# B&R Automation Studio project vibratorControlWithCurrentController (part 10)

#### local.typ - Local data types
```iecst
TYPE
	local_no_opcua_typ : 	STRUCT
		configOld : config_vibrator_typ;
		recipeOld : recipe_vibrator_typ;
		configTmp : config_vibrator_typ;
		axisAlarmText : STRING[363];
		alarm : local_alarm_typ;
		TON_alarmReaction : TON;
		calibration : local_no_opcua_calibration_typ;
	END_STRUCT;
	local_no_opcua_calibration_typ : 	STRUCT
		maxAmplitude : REAL;
		maxVibration : REAL;
		stepSizeAmplitude : REAL;
		tmpAmplitude : REAL;
		counter : USINT;
		bufferIdx : UINT;
		countTestPulse : USINT;
		boostCaliDone : BOOL;
		breakCaliDone : BOOL;
		countPulsesToFinetune : USINT;
	END_STRUCT;
	local_typ : 	STRUCT
		recipeName : STRING[80];
		configName : STRING[80];
		recipeNameCurrent : STRING[80];
		calibration : calibration_typ;
		MpRecipeRegPar_Config : MpRecipeRegPar;
		MpRecipeRegPar_Recipe : MpRecipeRegPar;
		MpRecipeRegPar_RecipeCurrent : MpRecipeRegPar;
		time : local_time_typ;
		MTBasicsLimiter_0 : MTBasicsLimiter;
		MC_BR_WriteParID_0 : MC_BR_WriteParID;
		vibAmplitude : REAL;
		highSpeed : BOOL;
		vibPercentAmplitude : REAL; (*amplitude for P3*)
		oldVibPercentAmplitude : REAL;
		vibAcceleration : REAL;
		sweep : local_sweep_typ;
		hmi : hmi_typ;
		vibFrequency : REAL := 50; (*[Hz] Frequency of virator*)
		calibrateState : UDINT;
		rampUp : REAL;
		linearizationSweep : linearizationSweep_typ;
		hw : local_hw_typ;
		linearizationTable : MTLookUpTable;
		lookUpFrequency : MTLookUpTable;
		pointsInLinearization : USINT;
		testAmplitude : BOOL;
		testDefault : BOOL;
		verifyLinearization : ARRAY[0..9]OF REAL;
		verifyIdx : USINT;
		testPercent : BOOL;
		oldSpeed : LEGO_SPEED_ENUM;
		oldCheckChangesConfig : BOOL;
		oldCheckChangesRecipe : BOOL;
		oldLoaded : BOOL;
		oldLoadedRecipe : BOOL;
		minimumTimeInCount : UDINT := 60000;
		DTGetTime_0 : DTGetTime;
		stateSimuPulse : USINT;
		simuTimeInCountSpeed : UDINT := 1000000;
		simuTimeInWaitSpeed : UDINT := 500000;
		simuTimeInStopped : UDINT := 600000;
		testProdFlow : BOOL;
		TON_delay : TON;
		currentAcceleration : REAL;
	END_STRUCT;
	calibration_typ : 	STRUCT
		TON_0 : TON;
		maxFreq : REAL;
		analogVib : REAL;
		sweepAmpl1CF : REAL := 0.5;
		sweepAmpl2CF : REAL := 0.6;
		sweepAmpl3CF : REAL := 1.0;
		sweepAmpl1LF : REAL := 0.09;
		sweepAmpl2LF : REAL := 0.08;
		sweepAmpl3LF : REAL := 0.11;
		sweepAmpl1LFbig : REAL := 0.1;
		sweepAmpl2LFbig : REAL := 0.08;
		sweepAmpl3LFbig : REAL := 0.11;
		sweepAmpl1CFbig : REAL := 1.7;
		sweepAmpl2CFbig : REAL := 1.4;
		sweepAmpl3CFbig : REAL := 1.8;
		timeToGetVibrWarm : TIME := T#11s;
		maxFreqFastSweep : REAL;
		bypassWarmUp : BOOL;
		slope : REAL;
		minAcceleration : REAL;
		minAccelerationTime : REAL;
		minAccelerationPhaseVelocity : REAL;
		accelerationStart : REAL;
		minAccelerationStart : REAL;
		freqBrakeCaliOffset : REAL;
		minFrequency : REAL;
		accelerationEnd : REAL;
		startBrakeFrequency : REAL;
	END_STRUCT;
	hmi_calibrate_typ : 	STRUCT
		activate : BOOL;
		calibrationToolPlugged : BOOL;
		progress : USINT;
		percentValue : REAL;
		testBoost : BOOL;
		enableStopButton : BOOL;
		runTestPulses : BOOL;
		increaseBoost : BOOL;
		increaseBrake : BOOL;
		decreaseBoost : BOOL;
		decreaseBrake : BOOL;
		enableBoostBrakeAdjustment : BOOL;
	END_STRUCT;
	linearizationSweep_typ : 	STRUCT
		actVibOld : REAL;
		sweepIdx : USINT;
		stableTime_TON : TON;
		a : REAL; (*Slope of linear function*)
		b : REAL; (*Intersection with y-axis in linear function*)
		MTBasicsPID_0 : MTBasicsPID;
		countStableSamples : USINT; (*If signal is less than allowed control error count one up.*)
		actIsOverSetValue : BOOL; (*True if act value is over set value.*)
		dcBusVoltage : REAL;
		supplyType : USINT; (*0=230V, 0=110V (Mexico)*)
	END_STRUCT;
	force_hw_typ : 	STRUCT
		enable : BOOL;
		current : REAL;
	END_STRUCT;
	hmi_typ : 	STRUCT
		config : config_vibrator_typ;
		calibratingProcessing : BOOL;
		cancelTuning : BOOL;
		recipe : recipe_vibrator_typ;
		calibration : hmi_calibrate_typ;
		force : force_hw_typ;
		needLinearization : BOOL;
		linearizationProcessing : BOOL;
		stopSweep : BOOL;
		oldCfType : SINT;
		actVoltage : REAL;
		targetAcceleration : REAL;
		voltage10Percent : REAL;
		voltage100Percent : REAL;
		recipeCurrent : recipe_vibrator_typ;
		waitSpeedLastBrick : USINT := 5;
		confirmPct : BOOL;
		increaseVibAmplitude : BOOL;
		decreaseVibAmplitude : BOOL;
		increaseVibAmplitudeFast : BOOL;
		decreaseVibAmplitudeFast : BOOL;
		linearizationGoalValue : REAL;
		enableOperatorInput : BOOL;
		showErrorMsgLinearization : BOOL;
		stopLinearization : BOOL;
		fitPercentTooLow : BOOL;
		linearizationActValue : REAL;
		daysSinceCalibration : REAL;
	END_STRUCT;
	local_time_typ : 	STRUCT
		elapsed : UDINT;
		maximum : UDINT;
	END_STRUCT;
	config_vibrator_typ : 	STRUCT
		tuneOnStartup : BOOL;
		vibFrequency : REAL := 50000;
		maxCurrent : REAL := 2.4;
		maxVoltage : REAL := 200;
		type : SINT; (*0=small CF, 1=big CF*)
		linearizationNodeVectorX : ARRAY[0..49]OF REAL;
		linearizationFcnValues : ARRAY[0..49]OF REAL;
		linearizationAccValues : ARRAY[0..49]OF REAL;
		linearizationFrequency1 : REAL; (*First frequency used for linear function for "voltage,frequency"*)
		linearizationFrequency2 : REAL; (*Second frequency used for linear function for "voltage,frequency"*)
		linearizationVoltage1 : REAL; (*First voltage used for linear function*)
		linearizationVoltage2 : REAL; (*Second voltage used for linear function*)
		pointY1 : REAL := 14;
		pointX1 : REAL := 10;
		pointY2 : REAL := 105;
		pointX2 : REAL := 100;
		Gain : REAL := 0.2;
		IntegrationTime : REAL := 1.5;
		minOut : REAL := 20;
		maxOut : REAL := 200;
		stableWindowPercent : REAL := 0.015;
		linearizeUsing3Points : BOOL := TRUE; (*True = only use 10%,55%,100% for linearization. *)
		frequencyVaryMode : BOOL := TRUE; (*This mode will vary the frequency depending on amplitude used on vibrator*)
		linearizationPercent : ARRAY[0..MAX_LOOKUP_POINTS]OF REAL;
		linearizationCurrent : ARRAY[0..MAX_LOOKUP_POINTS]OF REAL; (*Current at different percentages*)
		linearizationFrequencies : ARRAY[0..MAX_LOOKUP_POINTS]OF REAL; (*Frequency at different amplitudes*)
		linearizationAmplitude : ARRAY[0..MAX_LOOKUP_POINTS]OF REAL; (*Amplitude [A]*)
		fitPercentage : REAL; (*R^2 coefficient*)
		verifyLinearization : ARRAY[0..9]OF REAL;
		linearizationAccValue10pct : REAL;
		linearizationAccValue55pct : REAL;
		linearizationAccValue100pct : REAL;
		amplitudeFineTuning : REAL; (*This value will be add/subtract to the amplitude linearization result in case the calibration is a little off.*)
		emptyPercent : REAL;
		minimumTimeInCount : UDINT := 60000;
		calibrationDateTime : DATE_AND_TIME;
		boostVelocityLow : REAL;
		boostVelocityHigh : REAL;
		brakePhaseShiftVelocity : REAL;
		boostPhaseShiftVelocity : REAL;
		brakeVelocity : REAL;
		boostFrequency : REAL;
		brakeFrequency : REAL;
		boostAmplitude : REAL;
		brakeAmplitude : REAL;
		autoLinearizationAccAtCurrent : ARRAY[0..MAX_IDX_AUTO_LINEARIZATION]OF REAL;
		autoLinearizationCurrent : ARRAY[0..MAX_IDX_AUTO_LINEARIZATION]OF REAL;
		caliPulseBufferAcc : ARRAY[0..MAX_BUFFER_CALI_IDX]OF USINT;
		caliPulseEstimatedPct : ARRAY[0..MAX_BUFFER_CALI_IDX]OF USINT;
		disableLFBoost : BOOL;
	END_STRUCT;
	recipe_vibrator_typ : 	STRUCT
		waitSpeed : USINT := 10; (*%*)
		countingSpeed : USINT := 30; (*%*)
		rampUp : INT := 0; (*Time for 0 to 100 percent in msec*)
		useWaitSpeedCountingLastElement : BOOL := FALSE; (*If portion >2 and this is TRUE the vibrators will use waitSpeed when counting the last element, but belt will still keep counting speed.*)
	END_STRUCT;
	local_alarm_typ : 	STRUCT
		axisError : gAlarm_struct_typ;
	END_STRUCT;
	local_sweep_typ : 	STRUCT
		start : BOOL;
		amplitudeCFsmall : REAL := 0.8;
		amplitudeCFlarge : REAL := 1.2;
		amplitudeLF : REAL := 0.1;
		MTDataMinMax_0 : MTDataMinMax;
		frequencyStart : REAL := 48.5;
		frequencyStop : REAL := 50.4;
		maxVibrationISO : REAL;
		maxVibration : REAL;
		freqChangeRate : REAL := 0.02;
	END_STRUCT;
	local_hw_typ : 	STRUCT
		actVib : REAL;
		toggleBit : BOOL; (*Toggle bit will be true when we have new data ready*)
		ISO : REAL;
		analogInput : REAL;
		do_isBigCF : BOOL;
	END_STRUCT;
	axis_typ : 	STRUCT
		cmd : axis_cmd_typ;
		status : axis_status_typ;
		internal : axis_internal_typ;
	END_STRUCT;
	axis_cmd_typ : 	STRUCT
		power : BOOL;
	END_STRUCT;
	axis_status_typ : 	STRUCT
		powerOn : BOOL;
	END_STRUCT;
	axis_internal_typ : 	STRUCT
		MC_Power_0 : MC_Power;
	END_STRUCT;
	hmi_em_status_typ : 	STRUCT
		state : brdk_em_states_typ;
		substate : STRING[BRDK_MU_MAX_DESCRIPTION_STRING];
	END_STRUCT;
END_TYPE
```

#### local.var - Local variables
```iecst
VAR CONSTANT
	STATOR_RESISTANCE_SMALL_CF : REAL := 4.12;
	STATOR_RESISTANCE_SMALL_LF : REAL := 150;
	STATOR_INDUCTANCE_SMALL_CF : REAL := 0.230;
	STATOR_INDUCTANCE_SMALL_LF : REAL := 3.73;
	STATOR_RESISTANCE_BIG_CF : REAL := 4.96;
	STATOR_RESISTANCE_BIG_LF : REAL := 148.7;
	STATOR_INDUCTANCE_BIG_CF : REAL := 0.3;
	STATOR_INDUCTANCE_BIG_LF : REAL := 3.92;
	MAX_BUFFER_CALI_IDX : UINT := 399;
	VIBRATOR_FREQ_OFFSET : REAL := 0.1;
	VIBRATOR_FREQ_OFFSET_BIG_CF : REAL := 0.05;
END_VAR
VAR
	recipe : REFERENCE TO recipe_vibrator_typ;
	config : REFERENCE TO config_vibrator_typ;
	configTmp : REFERENCE TO config_vibrator_typ;
	em : REFERENCE TO brdkEM;
	i : UINT;
	j : USINT;
	k : UINT;
	localVariables : ARRAY[0..NUM_VIBRATOR] OF local_typ;
	localModule : ARRAY[0..NUM_VIBRATOR] OF brdkEM;
	this : REFERENCE TO local_typ;
	interface : REFERENCE TO gVibratorInterface_typ;
	watchIdx : USINT;
	axis : REFERENCE TO brdkMcBasic;
	localAxis : ARRAY[0..NUM_VIBRATOR] OF brdkMcBasic;
END_VAR
VAR CONSTANT
	MAX_IDX_AUTO_LINEARIZATION : USINT := 19;
	MAX_LOOKUP_POINTS : USINT := 4;
	SINE_WAVE_GENERATOR : UINT := 8752;
	CONTROLLER_MODE : UINT := 5;
	RATIO_ISO_TO_MAXPEAK : REAL := 95; (*Ration from ISO -> maxPeak (accelerometer value)*)
END_VAR
VAR
	em_status : ARRAY[0..NUM_VIBRATOR] OF hmi_em_status_typ;
	local : REFERENCE TO local_no_opcua_typ;
	local_no_opcua : ARRAY[0..NUM_VIBRATOR] OF local_no_opcua_typ;
END_VAR
```

#### LocalFunctions.fun
```iecst
{REDUND_ERROR} FUNCTION RSquared : REAL (*TODO: Add your comment here*) (*$GROUP=User,$CAT=User,$GROUPICON=User.png,$CATICON=User.png*)
	VAR_INPUT
		data : ARRAY[0..9] OF REAL;
		prc10 : REAL;
		prc100 : REAL;
	END_VAR
	VAR
		i : USINT;
		ssTot : REAL;
		ssRes : REAL;
		mean : REAL;
	END_VAR
END_FUNCTION

FUNCTION maxPeakToPercent : REAL
	VAR_INPUT
		maxPeakVal : REAL;
		Y1 : REAL;
		Y2 : REAL;
	END_VAR
	VAR
		slope : REAL;
	END_VAR
END_FUNCTION

FUNCTION getAccelerationFromPercent : REAL
	VAR_INPUT
		percent : REAL;
		vibratorType : UINT; (*0=CF, 1=LF*)
		machineType : SINT; (*0=small, 1=big*)
	END_VAR
END_FUNCTION
```

#### LocalFunctions.st
```iecst
FUNCTION RSquared
	mean := 0;
	FOR i:=0 TO 9 DO
		mean := mean + data[i];
	END_FOR
	mean := mean / 10;
	ssTot := 0;
	FOR i:=0 TO 9 DO
		ssTot := ssTot + pow(data[i]-mean, 2);
	END_FOR
	ssRes := 0;
	FOR i:=0 TO 9 DO
		ssRes := ssRes + pow(data[i]-(prc10+(((prc100-prc10)/9)*USINT_TO_REAL(i))), 2);
	END_FOR
	RSquared := 1 - (ssRes/ssTot);
END_FUNCTION

FUNCTION maxPeakToPercent
	IF (Y2-Y1) <> 0 THEN
		slope := 90/(Y2-Y1);
		maxPeakToPercent := LIMIT(0,slope*maxPeakVal+(10-(slope*Y1)),200);
	END_IF
END_FUNCTION

FUNCTION getAccelerationFromPercent

	IF machineType=0 THEN
		IF vibratorType=0 THEN
			// 10%=2756 , 100%=17420
			getAccelerationFromPercent := percent*162.93+1126.7;
		ELSE
			// 10%=1300 , 100%=10140
			getAccelerationFromPercent := percent*98.222+317.78;
		END_IF
	ELSE
		IF vibratorType=0 THEN
			// 10%=1456 , 100%=8060
			getAccelerationFromPercent := percent*73.378+722.22;
		ELSE
			// 10%=1508 , 100%=8840
			getAccelerationFromPercent := percent*81.467+693.33;
		END_IF
	END_IF

END_FUNCTION
```

### vibratorGlobal.typ
```iecst
TYPE
	gVibratorInterface_typ : 	STRUCT
		cmd : gVibratorInterface_cmd_typ;
		parameter : gVibratorInterface_parameter_typ;
		status : gVibratorInterface_status_typ;
	END_STRUCT;
	gVibratorInterface_cmd_typ : 	STRUCT
		speed : LEGO_SPEED_ENUM;
		calibrate : BOOL;
		copyRecipe : copy_recipe_command_typ;
		useWaitSpeed : BOOL; (*belt -> vibrator . Use waitSpeed even though belt is using countSpeed.*)
		monitorHighestAmplitude : BOOL; (*Will monitor highest analog acc value on accelerometer.*)
		readCurrentAndVoltage : BOOL;
		monitorActPeakValue : BOOL;
		monitorMaxPeakValue : BOOL;
		calibrationDone : BOOL;
		testPulses : BOOL;
		emptyPercent : REAL;
		reduceCountspeedWith5 : BOOL;
		runManualTest : BOOL;
		putRecipeForStalkElement : BOOL;
		initRecipe : BOOL;
		setCfType : BOOL;
	END_STRUCT;
	gVibratorInterface_parameter_typ : 	STRUCT
		speedPctManualTest : REAL;
		machineSize : USINT; (*0=Small CM, 1=Big CM*)
		CFType : USINT;
	END_STRUCT;
	gVibratorInterface_status_typ : 	STRUCT
		start : BOOL;
		calibrationDone : BOOL;
		calibratingMode : BOOL;
		machineType : SINT; (*0=small CM20, 1=big CM20*)
		highestAmplitudeAnalog : REAL;
		highestAmplitudeISO : REAL;
		highestAmplitudePeak : REAL;
		highestFrequencyAnalog : REAL;
		highestFrequencyISO : REAL;
		highestFrequencyPeak : REAL;
		highestAmplitude : REAL;
		highestFrequency : REAL;
		New_Member : USINT;
		actCurr : REAL;
		maxPeakValue : REAL;
		waitSpeed : USINT;
		countingSpeed : USINT;
		vibFrequency : REAL;
		vibAmplitude : REAL;
		vibAmplitudePercent : REAL;
		forcing : BOOL;
		percent : REAL;
		linearizationAmplitude : ARRAY[0..4]OF REAL;
		linearizationFrequencies : ARRAY[0..4]OF REAL;
		powered : BOOL;
		currAccelerometerPercent : REAL;
		currAccelerometerValue : REAL;
		calibrateBoost : BOOL;
		calibrateBrake : BOOL;
		brakePhaseShiftVelocity : REAL;
		boostPhaseShiftVelocity : REAL;
		minAccelerationStart : REAL;
		minAcceleration : REAL;
		minAccelerationTime : REAL;
		boostFrequency : REAL;
		brakeFrequency : REAL;
		brakeVelocity : REAL;
		boostVelocityLow : REAL;
		boostVelocityHigh : REAL;
		caliBoostVelocityLow : REAL;
		caliBoostVelocityHigh : REAL;
		calibrateBraketime : REAL;
		calibrateBrakeAmplitudeEnd : REAL;
		calibrateBrakeFrequencyEnd : REAL;
		boostAmpltiude : REAL;
		brakeAmplitude : REAL;
		caliProdTest : BOOL;
		currEstimatedPercent : REAL;
		isBigCF : BOOL;
		maxBoostPercent : REAL;
		minBreakPercent : REAL;
		filteredAccelerometerPercent : REAL;
		disableLFBoost : BOOL;
		rampUp : INT;
		calibrationResultFrequency : REAL;
		calibrationResultCurrent : REAL;
		calibrationResultCurrentOK : BOOL;
		calibrationResultFrequencyOK : BOOL;
		calibrationResultsReady : BOOL;
	END_STRUCT;
END_TYPE
```

### vibratorGlobal.var
```iecst
VAR
	gVibratorInterface : ARRAY[0..NUM_VIBRATOR] OF gVibratorInterface_typ;
END_VAR
VAR CONSTANT
	VIBRATOR_ALARM_SIZE : USINT := 0;
	NUM_VIBRATOR : USINT := 1; (*1 means 2*)
END_VAR
```

### Program Logical/modules/main/belt/belt (IEC)

#### producing.st
```iecst
ACTION producing:

	CASE em.state OF

		STATE_ACTIVATING:

			CASE em.substate OF

				0:
					IF (gRecipe.status.saved OR gRecipe.status.loaded) AND (gConfig.status.saved OR gConfig.status.loaded) THEN
						em.substate := 10;
					END_IF

				10:
					// Wait 20ms to make sure recipe is in the global variable. (belt in faster cyclic than vibrator)

					this.timeMinInCount := this.timeMinInCount + em.status.cycleTime;
					IF this.timeMinInCount > 20000 THEN
						this.timeMinInCount := 0;
						// Load CF/LF countspeed from recipe
						CFCountSpeed := gVibratorInterface[0].status.countingSpeed;
						LFCountSpeed := gVibratorInterface[1].status.countingSpeed;
						interface.status.recipeLoaded := TRUE;
						em.substate := 20;
					END_IF

				20:
					em.cmd.sc := TRUE;

			END_CASE

		STATE_STOPPED:
			em.description 	:= 'Waiting for start command';

			IF gConfig.status.loadInitialValue[2] AND (gRecipe.status.saved OR gRecipe.status.loaded) AND (gConfig.status.saved OR gConfig.status.loaded) THEN
				gConfig.status.loadInitialValue[2] := FALSE;
				recipe.countingSpeed := 300;
				recipe.useWaitSpeed := TRUE;
				recipe.waitSpeed := 110;
				recipe.rampUp := 50;
				recipe.rampDown := 30;
				recipe.itemGap := FALSE;
			END_IF

			// This case ONLY used for FAT
			CASE em.substate OF

				0:
					em.description := 'Wait for command';

					IF interface.cmd.doPhotoSensorTest THEN
						interface.status.photoSensorTestResult := TEST_NOT_DONE;
						this.hmi.statusFAT.torqueTestMaxProgress := 12000;
						this.hmi.statusFAT.torqueTestProgress := 0;
						this.hmi.statusFAT.photoSensorTestProgress := 0;
						this.hmi.statusFAT.photoSensorTestActive := TRUE;

						em.substate := 10;
					ELSIF interface.cmd.doPhotoSensorTestNoBelt THEN
						interface.cmd.doPhotoSensorTestNoBelt := FALSE;
						interface.status.photoSensorTestNoBeltResult := TEST_NOT_DONE;
						this.hmi.statusFAT.photoSensorTestNoBeltRunning := TRUE;
						this.timeElapsed := 0;
						em.substate := 50;
					END_IF

				10:
					em.description := 'Start servo and wait until it is running';

					interface.cmd.runManualTest := TRUE;
					interface.parameter.speedManualTest := 400;

//					IF this.hmi.cmd.stopPhotoSensorTest THEN	// stop cmd from user.
//						this.hmi.cmd.stopPhotoSensorTest := FALSE;
//						interface.status.photoSensorTestResult := TEST_STOPPED;
//						interface.cmd.startBelt := FALSE;
//						interface.par.beltSpeed := 0;
//						interface.cmd.doPhotoSensorTest := FALSE;
//						this.photoSensorTestProgress := 0;
//						this.hmi.status.photoSensorTestActive := FALSE;
//						em.substate := 0;
					IF axis.status.inMotion AND ABS(axis.status.actVelocity) > (interface.parameter.speedManualTest-50) THEN	// axis is running
						this.hmi.statusFAT.photoSensorTestProgress := 0;
						this.TON_photoSensorTest.PT := T#12000ms;
						this.TON_photoSensorTest.IN := FALSE;
						this.TON_photoSensorTest();
						// read parid for motor torque
						this.MC_BR_ReadParID_277.Axis := ADR(gAxisBelt);
						this.MC_BR_ReadParID_277.ParID := 277;
						this.MC_BR_ReadParID_277.DataType := ncPAR_TYP_REAL;
						this.MC_BR_ReadParID_277.DataAddress := ADR(this.motorTorque);
						this.MTDataMean_torque.Enable := TRUE;
						this.MTDataMean_torque.Reset := FALSE;
						this.MTDataMean_torque();

						em.substate := 11;
					END_IF

				11:
					em.description := 'Running photoSensor test';
					this.TON_photoSensorTest.IN := TRUE;
					// progress
					this.hmi.statusFAT.photoSensorTestProgress := TIME_TO_REAL(this.TON_photoSensorTest.ET);

					// read motor torque while running test.
					this.MC_BR_ReadParID_277.Execute := TRUE;
					this.MC_BR_ReadParID_277.Axis := ADR(gAxisBelt);
					this.MC_BR_ReadParID_277.DataAddress := ADR(this.motorTorque);

					IF this.MC_BR_ReadParID_277.Done THEN
						this.MC_BR_ReadParID_277.Execute := FALSE;
					END_IF
					this.MC_BR_ReadParID_277();
					IF this.hmi.statusFAT.photoSensorTestProgress >= 2500 THEN
						this.MTDataMean_torque.Reset := TRUE;
						this.MTDataMean_torque.In := ABS(this.motorTorque);
					END_IF
					this.MTDataMean_torque();

//					IF this.hmi.cmd.stopPhotoSensorTest THEN	// stop cmd from user.
//						this.hmi.cmd.stopPhotoSensorTest := FALSE;
//						this.TON_photoSensorTest.IN := FALSE;
//						interface.status.photoSensorTestResult := TEST_STOPPED;
//						interface.cmd.startBelt := FALSE;
//						interface.par.beltSpeed := 0;
//						interface.cmd.doPhotoSensorTest := FALSE;
//						this.photoSensorTestProgress := 0;
//						this.hmi.status.photoSensorTestActive := FALSE;
//						this.MTDataMean_torque(Enable:=FALSE,Reset:=FALSE);
//						em.substate := 15;
					IF this.hw.di_photo THEN
						interface.status.photoSensorTestResult := TEST_NOT_OK;
						this.TON_photoSensorTest.IN := FALSE;
						interface.cmd.runManualTest := FALSE;
						interface.parameter.speedManualTest := 0;
						this.hmi.avgMotorTorque := this.MTDataMean_torque.Out;
						interface.cmd.doPhotoSensorTest := FALSE;
						this.hmi.statusFAT.photoSensorTestProgress := 0;
						this.hmi.statusFAT.photoSensorTestActive := FALSE;
						this.MTDataMean_torque(Enable:=FALSE,Reset:=FALSE);
						em.substate := 15;
					ELSIF this.TON_photoSensorTest.Q THEN		// TODO: distanceConveyorShouldRun=6000 is random. How long should it run??
						IF this.MTDataMean_torque.Out < 0.25 THEN
							interface.status.photoSensorTestResult := TEST_OK;
							this.TON_photoSensorTest.IN := FALSE;
							interface.cmd.runManualTest := FALSE;
							interface.parameter.speedManualTest := 0;
							this.hmi.avgMotorTorque := this.MTDataMean_torque.Out;
							this.MTDataMean_torque(Enable:=FALSE,Reset:=FALSE);
							interface.cmd.doPhotoSensorTest := FALSE;
							this.hmi.statusFAT.photoSensorTestActive := FALSE;
							em.substate := 15;
						ELSE
							interface.status.photoSensorTestResult := TEST_NOT_OK;
							this.TON_photoSensorTest.IN := FALSE;
							interface.cmd.runManualTest := FALSE;
							this.hmi.avgMotorTorque := this.MTDataMean_torque.Out;
							interface.parameter.speedManualTest := 0;
							interface.cmd.doPhotoSensorTest := FALSE;
							this.hmi.statusFAT.photoSensorTestProgress := 0;
							this.hmi.statusFAT.photoSensorTestActive := FALSE;
							this.MTDataMean_torque(Enable:=FALSE,Reset:=FALSE);
							em.substate := 15;
						END_IF
					END_IF
					this.TON_photoSensorTest();

				15:
					em.description := 'Wait for readParId to be done (not busy)';

					this.MC_BR_ReadParID_277.Execute := FALSE;
					this.MC_BR_ReadParID_277.Axis := ADR(gAxisBelt);
					this.MC_BR_ReadParID_277.DataAddress := ADR(this.motorTorque);
					this.MC_BR_ReadParID_277();

					IF NOT this.MC_BR_ReadParID_277.Busy THEN
						em.substate := 0;
					END_IF

				50:
					em.description := 'Photo sensor test with no belt';

					this.timeElapsed := this.timeElapsed + em.status.cycleTime;

					IF this.timeElapsed > 20000000 THEN // 20s
						interface.status.photoSensorTestNoBeltResult := TEST_NOT_OK;
						interface.cmd.doPhotoSensorTestNoBelt := FALSE;
						this.hmi.statusFAT.photoSensorTestNoBeltRunning := FALSE;
						em.substate := 0;
					ELSIF this.hw.di_photo THEN
						interface.status.photoSensorTestNoBeltResult := TEST_OK;
						this.hmi.statusFAT.photoSensorTestNoBeltRunning := FALSE;
						interface.cmd.doPhotoSensorTestNoBelt := FALSE;
						em.substate := 0;
					END_IF

			END_CASE

			IF EDGENEG(interface.cmd.runManualTest)  THEN
				this.hmi.force.enable := FALSE;
			ELSIF interface.cmd.runManualTest THEN
				this.hmi.force.enable := TRUE;
				this.hmi.force.speed := interface.parameter.speedManualTest;
			END_IF

			this.hmi.status := 0;
			em.cmd.sc 		:= TRUE;

		STATE_RESETTING:

			this.TON_missingElements(IN := FALSE);
			this.hmi.force.enable := FALSE;
			this.teach.beltSpeed := 35;
			this.teach.attemptCount := 0;
			this.teach.TON_timeout(IN := FALSE);
			this.timeElapsed := 0;

			//set ramps for axis

			interface.status.speed	:= lego_speed_stop;

			CASE em.substate OF
				0:
					em.description := 'power on axis';

					IF axis.status.powerOn THEN
						axis.parameter.homePosition := 0;
						axis.parameter.homeMode := mcHOME_DIRECT;
						axis.command.home := TRUE;
						em.substate := 10;
					ELSE
						axis.command.power := TRUE;
					END_IF

				10:
					em.description := 'home axis axis';

					IF axis.status.isHomed AND axis.status.actPosition = 0 THEN
						axis.command.home := FALSE;
						em.cmd.sc := TRUE;
					END_IF
			END_CASE

		STATE_STARTING:

			interface.status.speed := lego_speed_stop;
			this.setSpeed := 0;
			brsmemset(ADR(this.distBetweenBricksFIFO),0,SIZEOF(this.distBetweenBricksFIFO)); // reset FIFO when starting.
			this.fifoIdx := 0;
			this.forceBeltToRun := FALSE;
			gVibratorInterface[0].cmd.useWaitSpeed := gVibratorInterface[1].cmd.useWaitSpeed := FALSE;
			IF this.hmi.brickLength<1 AND recipe.itemGap THEN // if no user input for brick length just set 20mm (some number).
				// Generate error?
				this.hmi.brickLength := 20;
			END_IF
			em.cmd.sc := TRUE;

		STATE_EXECUTE:

			CASE em.substate OF

				0:
					em.description := 'Waiting for command to run';

					IF interface.cmd.dropBrick THEN
						interface.status.speed := lego_speed_counting;
						this.timeMinInCount := 0;
						em.substate := 10;
					ELSIF interface.cmd.afterCount THEN
						interface.cmd.afterCount := FALSE;
						this.BrickCounter_0.Reset := TRUE;
						em.substate := 30;
					ELSIF this.BrickDetector_0.Out THEN
						interface.status.speed := lego_speed_stop;
					END_IF

				10:
					em.description := 'Counting portion';

					this.TON_missingElements.IN := TRUE;
					this.TON_missingElements.PT := T#10s;
					this.TON_missingElements();

					this.timeMinInCount := this.timeMinInCount + em.status.cycleTime; // Timer to latch lego_speed_count for min 1 cycle in 4.8ms (where vibrator is running) (we use UDINT because TON is not precise under 10ms)

					IF this.BrickCounter_0.Count >= interface.parameter.brickCountInPortion AND this.timeMinInCount >= 4800 THEN
						this.TON_missingElements.IN := FALSE;
						this.TON_missingElements();
						this.BrickCounter_0.Reset := TRUE;

						interface.status.speed := SEL(recipe.useWaitSpeed, lego_speed_stop, lego_speed_wait);
						em.substate := 20;
					END_IF

				20:
					em.description := 'Counting done';

					interface.status.dropBrickDone := TRUE;
					IF NOT interface.cmd.dropBrick THEN
						interface.status.dropBrickDone := FALSE;
						this.BrickCounter_0.Reset := FALSE;
						em.substate := 0;
					ELSIF this.BrickDetector_0.Out THEN
						interface.status.speed := lego_speed_stop;
					END_IF

				30:
					em.description := 'Handle aftercount';

					this.BrickCounter_0.Reset := FALSE;
					em.substate := 0;

			END_CASE

			// check what speeed to run
			CASE interface.status.speed OF
				lego_speed_stop:
					this.hmi.status := 1;
					this.setSpeed 	:= 0;

				lego_speed_counting:
					this.setSpeed := recipe.countingSpeed;
					this.hmi.status := 2;

				lego_speed_wait:
					this.hmi.status := 3;
					this.setSpeed := recipe.waitSpeed;

			END_CASE

			em.cmd.sc := TRUE;

		STATE_COMPLETING:

			CASE em.substate OF

				0:
					this.setSpeed := 0;
					interface.status.speed := lego_speed_stop;
					this.hmi.enableAutoMode := FALSE; // Disable automode if empty of machine is triggered.

					IF this.updateSpeedState=0 THEN
						this.SpeedRippleCalc_0.Enable := FALSE;
						this.SpeedRippleCalc_0();
						this.TON_speedRipple.IN := FALSE;
						this.TON_speedRipple();
						this.speedRippleChanged := FALSE;
						em.substate := 2;
					END_IF

				2:

					em.description := 'Emptying at max speed';

					IF interface.cmd.stopDoingEmpty THEN
						em.substate := 5;
					ELSE

						IF this.updateSpeedState=0 THEN	// only set speed when motionControl is rdy. Otherwise it might not be set.
							this.setSpeed := 500; // Max speed
						END_IF
						interface.status.speed := lego_speed_counting;

					END_IF

					IF interface.cmd.calibrate THEN
						em.substate := 10;
					END_IF

				5:
					em.description := 'Emptying - Waiting for wing to request brick';

					IF NOT interface.cmd.stopDoingEmpty THEN
						em.substate := 0;
					ELSE
						this.setSpeed := 0;
						interface.status.speed := lego_speed_stop;
					END_IF

					IF interface.cmd.calibrate THEN
						em.substate := 10;
					END_IF

				10:
					commonStoppingHoldingCompletingAbortingSuspending; // only run this action and em.cmd.sc = TRUE

			END_CASE

			// Meassure speed ripple doing emptiing
			this.TON_speedRipple.IN := axis.parameter.velocity=this.setSpeed AND NOT this.speedRippleChanged;
			this.TON_speedRipple.PT := T#10s;
			this.TON_speedRipple();

			this.SpeedRippleCalc_0.Enable := TRUE;
			this.SpeedRippleCalc_0.Axis := ADR(gAxisBelt);
			this.SpeedRippleCalc_0();

			IF this.TON_speedRipple.Q THEN
				this.TON_speedRipple.IN := FALSE;
				this.TON_speedRipple();

				config.speedRipple := this.SpeedRippleCalc_0.Out;
				this.speedRippleChanged := TRUE;
				this.SpeedRippleCalc_0.Enable := FALSE;
				this.SpeedRippleCalc_0();
			END_IF

		STATE_SUSPENDED:

			em.description := 'wing ready to receive drop';

			em.cmd.sc := TRUE;

		STATE_STOPPING, STATE_ABORTING, STATE_HOLDING,STATE_SUSPENDING:

			commonStoppingHoldingCompletingAbortingSuspending;

		STATE_ABORTED:

			this.hmi.status := 4;

			IF NOT MpAlarmXCheckReaction(mpAlarmXCore,'abortBelt') THEN
				em.cmd.sc := TRUE;
			END_IF

		STATE_CLEARING:

			commonClearing;

		ELSE

			em.cmd.sc := TRUE;

	END_CASE

END_ACTION
```

#### calibrating.st
```iecst
ACTION calibrating:

	CASE em.state OF

		STATE_STOPPED:

			IF this.abortedDoingTorqueTest THEN
				this.abortedDoingTorqueTest := FALSE;
				this.hmi.calibrating.activate := FALSE; //Should change to MODE_Production
			END_IF;
			em.cmd.sc := TRUE;

		STATE_RESETTING:

			IF this.hmi.calibrating.activate THEN
				interface.status.speed := lego_speed_stop;
				CASE em.substate OF
					0:
						em.description := 'power on axis';

						IF axis.status.powerOn THEN
							em.substate := 10;
						ELSE
							axis.command.power := TRUE;
						END_IF

					10:
						em.description := 'home axis axis';

						IF axis.status.isHomed THEN
							axis.command.home := FALSE;
							em.cmd.sc := TRUE;
						ELSE
							axis.command.home := TRUE;
						END_IF
				END_CASE
			ELSE
				em.cmd.sc := TRUE;
			END_IF

		STATE_STARTING:
			this.setSpeed := 0;
			this.abortedDoingTorqueTest := FALSE;
			interface.status.speed := lego_speed_stop;

			IF this.hmi.calibrating.activate THEN
				// motor torque
				this.MC_BR_ReadParID_277.Axis := ADR(gAxisBelt);
				this.MC_BR_ReadParID_277.ParID := 277;
				this.MC_BR_ReadParID_277.DataType := ncPAR_TYP_REAL;
				this.MC_BR_ReadParID_277.DataAddress := ADR(this.motorTorque);
			END_IF
			em.cmd.sc := TRUE;

		STATE_EXECUTE:
			IF this.hmi.calibrating.activate THEN
				// motor torque
				this.MC_BR_ReadParID_277.Execute := TRUE;
				this.MC_BR_ReadParID_277.Axis := ADR(gAxisBelt);
				this.MC_BR_ReadParID_277.DataAddress := ADR(this.motorTorque);

				IF this.MC_BR_ReadParID_277.Done THEN
					this.MC_BR_ReadParID_277.Execute := FALSE;
				END_IF

				this.MC_BR_ReadParID_277();
			END_IF

			CASE em.substate OF

				0:
					em.description := 'Only calibrate if it is for belt';

					em.cmd.sc := NOT this.hmi.calibrating.activate;

			END_CASE

			em.cmd.sc := TRUE;

		STATE_STOPPING, STATE_ABORTING, STATE_HOLDING:
			this.MTDataMean_torque(Enable := FALSE);
			this.MC_BR_ReadParID_277.Execute := FALSE;
			this.MC_BR_ReadParID_277();
			IF NOT this.MC_BR_ReadParID_277.Busy THEN
				commonStoppingHoldingCompletingAbortingSuspending;
			END_IF

		STATE_ABORTED:

			IF NOT MpAlarmXCheckReaction(mpAlarmXCore,'abortBelt') THEN
				em.cmd.sc := TRUE;
			END_IF

		STATE_CLEARING:
			this.hmi.avgMotorTorque := 0;
			this.abortedDoingTorqueTest := TRUE;
			commonClearing;

		ELSE

			em.cmd.sc := TRUE;

	END_CASE

END_ACTION
```

#### common.st
```iecst
ACTION commonStoppingHoldingCompletingAbortingSuspending:

	this.setSpeed := 0.0;
	interface.status.speed := lego_speed_stop;
	this.hmi.force.enable := FALSE;

	CASE em.substate OF
		0:
			em.description := 'If disabled it is stopped -> continue';

			IF axis.status.state <> DISABLED THEN
				em.substate := 5;		// go wait for axis to be stopped before taking power.
			ELSE
				em.cmd.sc := TRUE;
			END_IF

		5:
			em.description := 'waiting for belt to be stopped';

			IF NOT axis.status.inMotion THEN
				em.substate := 10;
			END_IF
		10:
			em.description := 'waiting for power of of servo axis';
			axis.command.power := FALSE;
			IF NOT axis.status.powerOn THEN
				em.cmd.sc := TRUE;
			END_IF
	END_CASE

END_ACTION

ACTION commonClearing:

	em.description := 'clear servo axis error(s)';

	IF axis.status.error.fault THEN
		axis.command.errorAcknowledge	:= TRUE;
	ELSE
		axis.command.errorAcknowledge	:= FALSE;
		brsmemset(ADR(this.alarm), 0, SIZEOF(this.alarm));
		//Set alarm texts
		this.alarm.missingElements.name := 'beltMissingElements';
		this.alarm.axisError.name := 'beltAxisError';
		this.alarm.beltBlocked.name := 'beltBlocked';
		em.cmd.sc := TRUE;
	END_IF

END_ACTION
```

#### motionControl.st
```iecst
ACTION motionControl:
	// Update speed on drive

	this.rampDown := 500/(UDINT_TO_REAL(MAX(1,recipe.rampDown+20))/1000);
	this.rampUp := 500/(UDINT_TO_REAL(MAX(1,recipe.rampUp+20))/1000);

	axis.parameter.acceleration	:= this.rampUp;
	axis.parameter.deceleration	:= this.rampDown;

	IF this.hmi.force.enable THEN
		axis.command.power := TRUE;
		IF(axis.status.powerOn) THEN
			IF axis.status.isHomed THEN
				axis.command.home := FALSE;
				axis.parameter.velocity		:= this.hmi.force.speed;
				IF NOT axis.status.inMotion OR this.hmi.force.speed <> this.oldForceSpeed THEN
					axis.command.moveVelocity	:= TRUE;
				ELSE
					axis.command.moveVelocity	:= FALSE;
				END_IF;
				this.oldForceSpeed := this.hmi.force.speed;
			ELSE
				axis.command.home := TRUE;
			END_IF

		ELSE
			axis.command.power := TRUE;
		END_IF
	ELSIF NOT this.hmi.force.enable AND this.hmi.force.enable <> this.oldForceActive THEN
		axis.command.power 			:= FALSE;
		axis.command.moveVelocity	:= FALSE;
	ELSIF em.mode = MODE_CALIBRATING THEN

		CASE this.updateSpeedState OF

			0:
				IF this.setSpeed <> this.speedOldManual THEN
					this.updateSpeedState := 10;
				END_IF
				this.speedOldManual := this.setSpeed;

			10:
				axis.parameter.velocity		:= this.setSpeed;
				axis.command.moveVelocity	:= TRUE;
				IF axis.status.done THEN	// When in motion .moveVelocity succeeded.
					this.updateSpeedState		:= 0;
					axis.command.moveVelocity	:= FALSE;
				END_IF

			20:
				axis.command.stop := TRUE;
				IF axis.status.stopped THEN
					axis.command.stop := FALSE;
					this.updateSpeedState := 0;
				END_IF

		END_CASE

	ELSE

		CASE this.updateSpeedState OF

			0:
				IF interface.status.speed <> this.speedOld THEN
					axis.parameter.velocity		:= this.setSpeed;
					axis.command.moveVelocity	:= TRUE;
					this.speedOld	:= interface.status.speed;
					this.oldPosition := axis.status.actPosition;
					this.updateSpeedState	:= 10;
				ELSIF em.state <> STATE_STARTING AND em.state <> STATE_EXECUTE AND interface.status.speed = 0 AND axis.status.inMotion THEN
					this.updateSpeedState := 20;
				END_IF

			10:
			//	IF axis.status.done OR interface.status.speed = lego_speed_stop OR (interface.status.speed = lego_speed_wait AND ) THEN	// When in motion .moveVelocity succeeded.
			//	IF axis.status.done OR interface.status.speed <> this.speedOld THEN	// When in motion .moveVelocity succeeded.
				IF axis.status.done OR interface.status.speed = lego_speed_stop OR (interface.status.speed = lego_speed_wait AND ABS(axis.status.actPosition-this.oldPosition) >= this.minMillimeterInCount) THEN
					this.updateSpeedState		:= 0;
					axis.command.moveVelocity	:= FALSE;
				END_IF

			20:
				axis.command.stop := TRUE;
				IF axis.status.stopped THEN
					axis.command.stop := FALSE;
					this.updateSpeedState := 0;
				END_IF

		END_CASE
	END_IF

	this.oldForceActive := this.hmi.force.enable;

	// torque limit control
	//this.MC_LimitLoad_0.Enable := axis.parameter.direction = this.MC_LimitLoad_0.Direction; // will call false for 1 scan if direction changes.
	//this.MC_LimitLoad_0.Axis := ADR(gAxisBelt);
	//this.MC_LimitLoad_0.Direction := axis.parameter.direction;
	//this.MC_LimitLoad_0.Load := config.maxTorqueAllowed;

	// Axis direction and torque limit
	CASE this.stateAxisDirection OF

		0:
		//	'Wait for config';

			IF gConfig.status.loaded THEN
				this.MC_BR_WriteParID_0(Execute := FALSE);
				this.oldMachineType := 99;
				this.stateAxisDirection := 10;
			END_IF

		10:
			this.TON_testDelay.IN := TRUE;
			this.TON_testDelay.PT := T#300ms;
			this.TON_testDelay();

			IF this.TON_testDelay.Q THEN
				this.TON_testDelay.IN := FALSE;
				this.TON_testDelay();

				this.stateAxisDirection := 15;
			END_IF

		15:
			// Wait to see if machineType changes.

			IF gMainInterface.status.machineType <> this.oldMachineType THEN
				this.oldMachineType := gMainInterface.status.machineType;

				this.stateAxisDirection := 20;
			END_IF

		20:
		//	'Set count_dir to inverse';

			this.MC_BR_WriteParID_0.Execute 		:= TRUE;
			this.MC_BR_WriteParID_0.Axis 			:= ADR(gAxisBelt);
			this.MC_BR_WriteParID_0.ParID 			:= 96; 					// Encoder1: Load scaling: Count direction
			this.MC_BR_WriteParID_0.DataType 		:= ncPAR_TYP_USINT;
			this.MC_BR_WriteParID_0.DataAddress 	:= SEL(this.oldMachineType=0,ADR(ncSTANDARD),ADR(ncINVERSE));
			this.MC_BR_WriteParID_0();

			IF this.MC_BR_WriteParID_0.Done THEN
				this.MC_BR_WriteParID_0(Execute := FALSE);
				this.MC_LimitLoad_0(Enable := FALSE);
				this.stateAxisDirection := 100;
			END_IF

		100:
			this.MC_LimitLoad_0.Axis := ADR(gAxisBelt);
			this.MC_LimitLoad_0.Direction := SEL(this.oldMachineType=0,0,1);
			this.MC_LimitLoad_0.Load := config.maxTorqueAllowed;
			this.MC_LimitLoad_0.Enable := TRUE;

			IF this.MC_LimitLoad_0.Ready THEN
				this.stateAxisDirection := 15;
			END_IF

	END_CASE

END_ACTION
```

#### alarm.st
```iecst
ACTION alarm:

	// Extra check if belt is stopped and vibrator is running. Happend in production
	IF (gVibratorInterface[0].status.percent > 0 OR gVibratorInterface[1].status.percent > 0) AND axis.status.actVelocity < 10.0 THEN
		this.timeBeltStoppedButVibrRunning := this.timeBeltStoppedButVibrRunning + em.status.cycleTime;
	ELSE
		this.timeBeltStoppedButVibrRunning := 0;
	END_IF

	// Missing elements
	this.alarm.missingElements.active := this.TON_missingElements.Q;
	IF this.alarm.missingElements.active AND NOT this.alarm.missingElements.oldActive THEN
		this.alarm.missingElements.instanceID := MpAlarmXSet(mpAlarmXCore, this.alarm.missingElements.name);
	ELSIF NOT this.alarm.missingElements.active AND this.alarm.missingElements.oldActive THEN
		MpAlarmXAcknowledgeID(mpAlarmXCore, this.alarm.missingElements.instanceID);
	END_IF
	this.alarm.missingElements.oldActive := this.alarm.missingElements.active;

	// Axis error alarm
	this.alarm.axisError.active := (axis.status.error.fault AND axis.status.driveStatus.initialized);
	IF this.alarm.axisError.active AND NOT this.alarm.axisError.oldActive THEN
		IF axis.status.error.count < 1 THEN
			this.alarm.axisError.instanceID := MpAlarmXSet(mpAlarmXCore, this.alarm.axisError.name);
		ELSE
			FOR j:=0 TO (axis.status.error.count-1) DO
				IF brdkStrSearch(ADR(axis.status.error.text.active[j]),ADR('Lag error')) <> -1 THEN
					this.alarm.beltBlocked.instanceID := MpAlarmXSet(mpAlarmXCore, this.alarm.beltBlocked.name);
					EXIT;
				ELSIF j=(axis.status.error.count-1) THEN
					this.alarm.axisError.instanceID := MpAlarmXSet(mpAlarmXCore, this.alarm.axisError.name);
				END_IF
			END_FOR
		END_IF
	END_IF
	this.alarm.axisError.oldActive := this.alarm.axisError.active;

	this.TON_alarmReaction.IN := TRUE;
	this.TON_alarmReaction.PT := T#200ms;
	this.TON_alarmReaction();

	IF this.TON_alarmReaction.Q THEN
		this.TON_alarmReaction.IN := FALSE;
		this.TON_alarmReaction();
		this.hmi.showHighWaitspeedAlarm := recipe.waitSpeed>140;
		this.hmi.enableStaticMode := NOT this.hmi.enableAutoMode;
		this.hmi.showPermanentAutoModeButton := NOT config.hideExperimentalFeatures;

		(****************************** REACTION ******************************)

		IF em.state <> STATE_ABORTED AND em.state <> STATE_ABORTING AND em.state <> STATE_CLEARING THEN
			IF MpAlarmXCheckReaction(mpAlarmXCore,'abortBelt') THEN
				em.cmd.abort := TRUE;
			END_IF
		END_IF
		(**********************************************************************)

	END_IF

END_ACTION
```

#### belt.st - Init, cyclic, exit code
```iecst
PROGRAM _INIT

	em.setup.name := 'belt';
	em.setup.parent.name := 'main';
	em.setup.lastActivated := FALSE;

	// gets the task name and setup names for config and receipe types
	ST_name(0,ADR(this.configName),0);
	brdkStrCpy(ADR(this.recipeName),ADR(this.configName));
	brdkStrCpy(ADR(this.recipeNameCurrent),ADR(this.configName));
	brdkStrCat(ADR(this.configName),ADR(':this.hmi.config'));
	brdkStrCat(ADR(this.recipeName),ADR(':this.hmi.recipe'));
	brdkStrCat(ADR(this.recipeNameCurrent),ADR(':this.hmi.recipeCurrent'));

	setupPointers;

	//=====================================================================================
	//						Axis adr setup
	//=====================================================================================
	axis.configuration.ignoreSwLimit	:= TRUE;
	axis.configuration.disableTemperatureReading := TRUE;
	axis.configuration.disableTorqueReading := TRUE;
	axis.configuration.disableLagErrorReading := TRUE;
	axis.configuration.period := 0;
	axis.configuration.factor := 100;

	//Set alarm texts
	this.alarm.missingElements.name := 'beltMissingElements';
	this.alarm.axisError.name := 'beltAxisError';
	this.alarm.beltBlocked.name := 'beltBlocked';

END_PROGRAM

PROGRAM _CYCLIC

	setupPointers;

	IF gMainInterface.status.simulation OR gSimulation.status.simulateAllButWing THEN
		this.hw.di_photo := gSimulation.status.photoSensor;
	END_IF

	//***********************************
	//          Brick Detector
	//***********************************
	this.BrickDetector_0.Signal 		:= this.hw.di_photo;
	this.BrickDetector_0.BeltPosition 	:= axis.status.actPosition;
	this.BrickDetector_0.ItemGap 		:= recipe.itemGap;
	this.BrickDetector_0.FlickeringFilterGap := config.flickeringFilterGap;
	this.BrickDetector_0.FlickeringFilterGapLong := config.flickeringFilterGapLong;
	this.BrickDetector_0();

	this.brickDetected := this.BrickDetector_0.Out;
	this.hmi.itemGapTeaching := this.BrickDetector_0.Teaching;

	//***********************************
	//          Brick Counter
	//***********************************
	this.BrickCounter_0.Signal 			:= this.BrickDetector_0.Out;
	this.BrickCounter_0();

	//***********************************
	//         Brick Information
	//***********************************
	this.BrickInfo_0.Signal 		:= this.BrickDetector_0.Out;
	this.BrickInfo_0.Speed 			:= interface.status.speed;
	this.BrickInfo_0.BeltPosition 	:= axis.status.actPosition;
	this.BrickInfo_0();

	this.hmi.avgDistanceBetweenBricks := this.BrickInfo_0.BrickGap;

	//***********************************
	// Ramp Up Time Calc
	//***********************************
//	this.RampUpTimeCalc_0.Enable := TRUE;
//	this.RampUpTimeCalc_0.BeltFeederSensor := NOT gFeederInterface.status.beltFeederEmpty;
//	this.RampUpTimeCalc_0.ChangeOverCounter := this.changeOverCounter;
//	this.RampUpTimeCalc_0.OKPortions := gUpperFlapInterface.status.OKPortions;
//	this.RampUpTimeCalc_0.Running := em.state = STATE_STARTING OR em.substate = STATE_EXECUTE;
//	this.RampUpTimeCalc_0.CFSensor := NOT gFeederInterface.status.vibratorBowlEmpty;
//	this.RampUpTimeCalc_0();
//
//	this.hmi.rampUpTime := this.RampUpTimeCalc_0.RampUpTime;

	//***********************************
	// Vibrator Controller (Auto Mode)
	//***********************************

	CASE interface.parameter.brickCountInPortion OF

		0,1:
			this.CFController_0.BrickGapTargetMin := 55;
			this.CFController_0.BrickGapTargetMax := config.brickGapCfMax1Portion;
			this.LFController_0.BrickGapTargetMin := config.brickGapLfMin1Portion;
			this.LFController_0.BrickGapTargetMax := 70;

		2:
			this.CFController_0.BrickGapTargetMin := 55;
			this.CFController_0.BrickGapTargetMax := config.brickGapCfMax2Portion;
			this.LFController_0.BrickGapTargetMin := config.brickGapLfMin2Portion;
			this.LFController_0.BrickGapTargetMax := 45;

		3:
			this.CFController_0.BrickGapTargetMin := 50;
			this.CFController_0.BrickGapTargetMax := config.brickGapCfMax3Portion;
			this.LFController_0.BrickGapTargetMin := config.brickGapLfMin3Portion;
			this.LFController_0.BrickGapTargetMax := config.brickGapLfMin3Portion;

		4:
			this.CFController_0.BrickGapTargetMin := config.brickGapCfMax4Portion;
			this.CFController_0.BrickGapTargetMax := config.brickGapCfMax4Portion;
			this.LFController_0.BrickGapTargetMin := config.brickGapLfMin4Portion;
			this.LFController_0.BrickGapTargetMax := config.brickGapLfMin4Portion;

		ELSE
			this.CFController_0.BrickGapTargetMin := config.brickGapCfMax4Portion;
			this.CFController_0.BrickGapTargetMax := config.brickGapCfMax4Portion;
			this.LFController_0.BrickGapTargetMin := config.brickGapLfMin4Portion;
			this.LFController_0.BrickGapTargetMax := config.brickGapLfMin4Portion;

	END_CASE

	// One time set belt speed in AutoMode when 20 bricks has been counted (If brick is very long a 2 portion might need to use same belt speed as a 4 portion small brick).
//	IF this.hmi.enableAutoMode AND this.BrickInfo_0.BrickCount=20 THEN
//		this.portionLength := (this.BrickInfo_0.BrickLength+this.LFController_0.BrickGapTargetMax)*UDINT_TO_REAL(interface.parameter.brickCountInPortion);
//
//		IF this.portionLength < 120 THEN
//			recipe.countingSpeed := 380;
//		ELSIF this.portionLength < 170 THEN
//			recipe.countingSpeed := 400;
//		ELSE
//			recipe.countingSpeed := 420;
//		END_IF
//	END_IF

	this.CFController_0.Enable := this.hmi.enableAutoMode;
	this.CFController_0.BrickGap := this.BrickInfo_0.BrickGap75;
	this.CFController_0.MaxOutput := SEL(this.BrickInfo_0.BrickLength=0, MIN(this.BrickInfo_0.BrickLength*2.5, 80), 80);
	this.CFController_0.PortionCount := interface.parameter.brickCountInPortion;
	this.CFController_0.Running := gVibratorInterface[0].status.percent > 0 AND (em.state = STATE_EXECUTE OR em.state = STATE_STARTING);
	this.CFController_0.NoElements := gFeederInterface.status.vibratorBowlEmpty;
	this.CFController_0.BeltMissingElements := this.BrickInfo_0.MissingElements AND em.state <> STATE_STOPPED;
	this.CFController_0.StaticOut := CFCountSpeed;
	this.CFController_0();

	this.LFController_0.Enable := this.hmi.enableAutoMode;
	this.LFController_0.BrickGap := this.BrickInfo_0.MinBrickGap;
	this.LFController_0.Running := gVibratorInterface[1].status.percent > 0 AND (em.state = STATE_EXECUTE OR em.state = STATE_STARTING);
	this.LFController_0.BeltMissingElements := this.BrickInfo_0.MissingElements AND em.state <> STATE_STOPPED;
	this.LFController_0.StaticOut := LFCountSpeed;
	this.LFController_0();

	this.CFController_0.LFOut := this.LFController_0.Out;

	IF this.LFController_0.Active THEN
		interface.status.LFCountSpeed := LIMIT(5,this.LFController_0.Out,130);
		interface.status.CFCountSpeed := LIMIT(10,this.CFController_0.Out,100);

		CFCountSpeed := interface.status.CFCountSpeed;
		LFCountSpeed := interface.status.LFCountSpeed;
	ELSE
		interface.status.CFCountSpeed := CFCountSpeed;
		interface.status.LFCountSpeed := LFCountSpeed;
	END_IF

	// Auto disable AutoMode if output is good!
	IF this.hmi.enableAutoMode THEN

		// Minimum wait 20 portions in EXECUTE before auto disabling
		IF interface.cmd.cycleTimeCount > 19 THEN

			CASE interface.parameter.brickCountInPortion OF

			0,1:
				IF gCapconInterface.status.cycleTimeAutoMode > config.cycleTimeToStopAutoMode1 THEN
					this.hmi.enableAutoMode := FALSE;
				END_IF

			2:
				IF gCapconInterface.status.cycleTimeAutoMode > config.cycleTimeToStopAutoMode2 THEN
					this.hmi.enableAutoMode := FALSE;
				END_IF

			3:
				IF gCapconInterface.status.cycleTimeAutoMode > config.cycleTimeToStopAutoMode3 THEN
					this.hmi.enableAutoMode := FALSE;
				END_IF

			4:
				IF gCapconInterface.status.cycleTimeAutoMode > config.cycleTimeToStopAutoMode4 THEN
					this.hmi.enableAutoMode := FALSE;
				END_IF

			ELSE
				IF gCapconInterface.status.cycleTimeAutoMode > config.cycleTimeToStopAutoMode4 THEN
					this.hmi.enableAutoMode := FALSE;
				END_IF

			END_CASE

		END_IF

	ELSIF NOT this.changeOverTriggered THEN
		interface.cmd.cycleTimeCount := 0;
	END_IF

	IF config.enablePermanentAutoMode THEN
		this.hmi.enableAutoMode := TRUE;
	END_IF

	IF this.changeOverTriggered THEN

		// After changeover wait 10 portions -> if output is low enable AutoMode
		IF interface.cmd.cycleTimeCount > 9 THEN
			this.changeOverTriggered := FALSE;

			CASE interface.parameter.brickCountInPortion OF

				0,1:
					IF gCapconInterface.status.cycleTimeAutoMode < config.cycleTimeToStopAutoMode1 THEN
						this.hmi.enableAutoMode := TRUE;
					END_IF

				2:
					IF gCapconInterface.status.cycleTimeAutoMode < config.cycleTimeToStopAutoMode2 THEN
						this.hmi.enableAutoMode := TRUE;
					END_IF

				3:
					IF gCapconInterface.status.cycleTimeAutoMode < config.cycleTimeToStopAutoMode3 THEN
						this.hmi.enableAutoMode := TRUE;
					END_IF

				4:
					IF gCapconInterface.status.cycleTimeAutoMode < config.cycleTimeToStopAutoMode4 THEN
						this.hmi.enableAutoMode := TRUE;
					END_IF

				ELSE
					IF gCapconInterface.status.cycleTimeAutoMode < config.cycleTimeToStopAutoMode4 THEN
						this.hmi.enableAutoMode := TRUE;
					END_IF

			END_CASE

		END_IF

		// If operator changes CountSpeeds don't auto trigger enableAutoMode. We believe that operator will tune the machine and don't want to trigger AutoMode in the middle of his work.
		IF CFCountSpeed <> gVibratorInterface[0].status.countingSpeed OR LFCountSpeed <> gVibratorInterface[1].status.countingSpeed THEN
			this.changeOverTriggered := FALSE;
		END_IF

	END_IF

	// TEMP FIX BECAUSE BIG BOWL HASNT BEEN IMPLEMENTED YET
	IF gVibratorInterface[0].parameter.machineSize = 1 THEN
		this.hmi.enableAutoMode := FALSE;
	END_IF

	CASE em.mode OF
		MODE_PRODUCING: producing;
		MODE_CALIBRATING: calibrating;
		ELSE em.cmd.sc := TRUE;
	END_CASE

	alarm;

	em();

	motionControl;
	this.MC_LimitLoad_0();
	axis();

	interface.status.calibratingMode := this.hmi.calibrating.activate;
	interface.status.actualPosition := ABS(axis.status.actPosition);
	interface.status.autoMode := this.hmi.enableAutoMode;

	// copy the recipe data
	CASE interface.cmd.copyRecipe OF

		COPY_RECIPE_NEXT_TO_WORKING:
			this.hmi.recipe 			:= this.hmi.recipeCurrent;
			gRecipe.cmd.save 			:= TRUE;
			this.changeOverCounter 		:= this.changeOverCounter + 1;
//			this.BrickInfo_0.Reset := TRUE;
//			this.BrickInfo_0();
//			this.LFController_0.Enable := FALSE;
//			this.LFController_0();
//			CFCountSpeed := 20;
//			LFCountSpeed := 40;
			interface.cmd.copyRecipe 	:= COPY_RECIPE_NONE;

		COPY_RECIPE_SANDBOX_TO_NEXT:
			interface.cmd.copyRecipe 	:= COPY_RECIPE_NONE;

	END_CASE

	// ----------------------- TODO TEST THIS !!!! ------------------------------------
	// vibrator -> belt. We have changeover and recipe values has been updated. Init with recipe parameters and reset VibratorController.
	IF interface.cmd.changeover THEN
		interface.cmd.changeover := FALSE;

		CFCountSpeed := gVibratorInterface[0].status.countingSpeed;
		LFCountSpeed := gVibratorInterface[1].status.countingSpeed;
		this.BrickInfo_0.Reset := TRUE;
		this.BrickInfo_0();
		this.CFController_0.Enable := FALSE;
		this.CFController_0();
		this.LFController_0.Enable := FALSE;
		this.LFController_0();
		IF gVibratorInterface[0].parameter.machineSize <> 1 AND config.enableAutoModeFeature THEN // Not Big Machine and auto mode enabled
			gCapconInterface.status.cycleTimeAutoMode := 0;
			interface.cmd.cycleTimeCount := 0; // to make sure we don't disable autoMode right aways
			this.CFController_0.LFOffset := LIMIT(0,LFCountSpeed-CFCountSpeed,10); // use the offset from recipe but limit it.
			this.changeOverTriggered := TRUE;
		END_IF
	END_IF

	IF interface.cmd.initRecipe THEN
		interface.cmd.initRecipe := FALSE;

		recipe.countingSpeed := LIMIT(350,recipe.countingSpeed,450);
		recipe.waitSpeed := LIMIT(100,recipe.waitSpeed,150);
		recipe.rampUp := 100;
		recipe.rampDown := 30;
	ELSIF interface.cmd.putRecipeForStalkElement THEN
		interface.cmd.putRecipeForStalkElement := FALSE;

		recipe.rampUp := 100;
		recipe.rampDown := 0;
		recipe.countingSpeed := 440;
		recipe.waitSpeed := 120;
		recipe.useWaitSpeed := TRUE;
	END_IF

	IF gRecipe.status.doCheckForChanges AND NOT this.oldCheckChangesRecipe THEN
		// chek if it has been loade then update old
		this.MpRecipeRegPar_Recipe.Enable := TRUE;
		this.MpRecipeRegPar_RecipeCurrent.Enable := TRUE;

		IF gRecipe.status.loaded AND NOT this.oldLoadedRecipe THEN
			// Initial program load. Set old=new to avoid saving just after a load (makes no sense)
			this.recipeOld := this.hmi.recipe;
		END_IF
		this.oldLoadedRecipe := gRecipe.status.loaded;

		IF NOT gRecipe.cmd.save AND gRecipe.status.loaded AND (brsmemcmp(ADR(this.hmi.recipe),ADR(this.recipeOld),SIZEOF(this.recipeOld)) <> 0) THEN
			gRecipe.cmd.save := TRUE;
			this.recipeOld := this.hmi.recipe;
		END_IF

	END_IF
	this.MpRecipeRegPar_Recipe(MpLink := ADR(mpRecipe), PVName := ADR(this.recipeName), Category := ADR('recipe'));
	this.MpRecipeRegPar_RecipeCurrent(MpLink := ADR(mpRecipeCurrent), PVName := ADR(this.recipeNameCurrent), Category := ADR('recipeCurrent'));
	this.oldCheckChangesRecipe := gRecipe.status.doCheckForChanges;

	IF gConfig.status.doCheckForChanges AND NOT this.oldCheckChangesConfig THEN
		this.MpRecipeRegPar_Config.Enable := TRUE;

		IF gConfig.status.loaded AND NOT this.oldLoaded THEN
			// Initial program load. Set old=new to avoid saving just after a load (makes no sense)
			this.configOld := this.hmi.config;
		END_IF
		this.oldLoaded := gConfig.status.loaded;

		IF NOT gConfig.cmd.save AND gConfig.status.loaded AND (brsmemcmp(ADR(this.hmi.config),ADR(this.configOld),SIZEOF(this.configOld)) <> 0) THEN
			gConfig.cmd.save := TRUE;
			this.configOld := this.hmi.config;
		END_IF

	END_IF
	this.MpRecipeRegPar_Config(MpLink := ADR(mpRecipe), PVName := ADR(this.configName), Category := ADR('config'));
	this.oldCheckChangesConfig := gConfig.status.doCheckForChanges;

	IF axis.status.error.fault THEN
		this.alarm.axisError.active	:= TRUE;
	ELSE
		this.alarm.axisError.active	:= FALSE;
	END_IF

	IF gConfig.status.factoryReset[2] THEN
		gConfig.status.factoryReset[2] := FALSE;
		// Factory reset all parameters:
		config.maxTorqueAllowed := 0.7; //0.7nm
	END_IF

	this.hmi.waitSpeedDisabled := NOT recipe.useWaitSpeed;

END_PROGRAM

PROGRAM _EXIT

	this.MpRecipeRegPar_Recipe(Enable := FALSE);
	this.MpRecipeRegPar_Config(Enable := FALSE);
	this.MpRecipeRegPar_RecipeCurrent(Enable := FALSE);

	this.MTDataMean_torque(Enable := FALSE);
	this.MC_LimitLoad_0(Enable := FALSE);
	this.MTBasicsLimiter_0(Enable := FALSE);

END_PROGRAM
```

#### setupPointers.st
```iecst
ACTION setupPointers:
	recipe ACCESS ADR(this.hmi.recipe);
	config ACCESS ADR(this.hmi.config);
	interface ACCESS ADR(gBeltInterface);
	axis.configuration.axis				:= ADR(gAxisBelt);
END_ACTION
```

#### FAT.st
```iecst
ACTION FAT:

END_ACTION
```

#### local.typ - Local data types
```iecst
TYPE
	local_teach_typ : 	STRUCT
		beltBackwardSpeed : INT := -40;
		beltSpeed : INT;
		beltBackwardTimeout : UDINT := 3000;
		capconTimeout : UDINT := 1500;
		attemptCount : USINT;
		TON_timeout : TON;
	END_STRUCT;
	hmi_calibrating_typ : 	STRUCT
		savePwmValueFor0mmPerSec : BOOL;
		savePwmValueFor100mmPerSec : BOOL;
		savePwmValueFor300mmPerSec : BOOL;
		savePwmValueFor500mmPerSec : BOOL;
		activate : BOOL;
		pwmValue : REAL;
		setSpeed : REAL := 200;
	END_STRUCT;
	hmi_force_hw_typ : 	STRUCT
		PWM : REAL;
		speed : REAL;
		enable : BOOL;
	END_STRUCT;
	local_typ : 	STRUCT
		TON_missingElements : TON;
		setSpeed : REAL; (*speed in mm/s*)
		oldSpeed : REAL; (*speed in mm/s*)
		actualSpeed : REAL; (*speed in mm/s*)
		pwmSpeed : REAL; (*converted speed from mm/s to pwm value %*)
		alarm : local_alarm_typ;
		hw : local_hw_typ;
		limiterState : USINT;
		configName : STRING[80];
		recipeName : STRING[80];
		recipeNameCurrent : STRING[80];
		MpRecipeRegPar_Config : MpRecipeRegPar;
		MpRecipeRegPar_Recipe : MpRecipeRegPar;
		MpRecipeRegPar_RecipeCurrent : MpRecipeRegPar;
		MTBasicsLimiter_0 : MTBasicsLimiter;
		highSpeed : BOOL;
		teach : local_teach_typ;
		configOld : config_belt_typ;
		recipeOld : recipe_belt_typ;
		hmi : hmi_typ;
		TON_stopDelay : TON;
		TON_startDelay : TON;
		rampDown : REAL;
		rampUp : REAL;
		currentCount : UDINT;
		updateSpeedState : USINT;
		speedOld : LEGO_SPEED_ENUM;
		speedOldManual : REAL;
		oldForceSpeed : REAL;
		oldForceActive : BOOL;
		capconNoStopDelay : UDINT; (*Time for no stop delay in capcon config*)
		MC_BR_ReadParID_277 : MC_BR_ReadParID; (*Motor torque*)
		motorTorque : REAL;
		MTDataMean_torque : MTDataMean;
		timeElapsed : UDINT;
		MC_LimitLoad_0 : MC_LimitLoad;
		abortedDoingTorqueTest : BOOL;
		distBetweenBricksFIFO : ARRAY[0..9]OF REAL; (*10 values in FIFO.*)
		previousEncPos : REAL;
		fifoIdx : USINT;
		distanceMovedSinceHighSignal : REAL;
		actPosAfterLastBrickInPortion : REAL; (*Position of axis after the last brick in portion (used to make sure that axis move a certain distance before stopping).*)
		forceBeltToRun : BOOL; (*Will force belt to run*)
		TON_alarmReaction : TON;
		brickDetected : BOOL;
		BrickDetector_0 : BrickDetector;
		BrickInfo_0 : BrickInfo;
		BrickCounter_0 : BrickCounter;
		oldDropBrick : BOOL;
		oldCheckChangesConfig : BOOL;
		oldCheckChangesRecipe : BOOL;
		oldLoaded : BOOL;
		oldLoadedRecipe : BOOL;
		axisAlarmText : STRING[363];
		RampUpTimeCalc_0 : RampUpTimeCalc;
		changeOverCounter : UDINT;
		timeBeltStoppedButVibrRunning : UDINT;
		oldPosition : LREAL;
		minMillimeterInCount : LREAL := 8.0;
		timeMinInCount : UDINT;
		SpeedRippleCalc_0 : SpeedRippleCalc;
		speedRippleChanged : BOOL;
		TON_speedRipple : TON;
		CFController_0 : CFController;
		LFController_0 : LFController;
		MC_BR_WriteParID_0 : MC_BR_WriteParID;
		TON_testDelay : TON;
		stateAxisDirection : USINT;
		oldMachineType : USINT;
		GetBrickGapTargetMinMax_0 : GetBrickGapTargetMinMax;
		portionLength : REAL;
		changeOverTriggered : BOOL;
		TON_photoSensorTest : TON;
	END_STRUCT;
	hmi_typ : 	STRUCT
		calibrating : hmi_calibrating_typ;
		config : config_belt_typ;
		recipe : recipe_belt_typ;
		mode : LEGO_SPEED_ENUM;
		status : USINT;
		statusFAT : hmi_status_FAT_typ;
		force : hmi_force_hw_typ;
		recipeCurrent : recipe_belt_typ;
		avgMotorTorque : REAL;
		waitSpeedDisabled : BOOL; (*Used for a warning if wait speed is disabled*)
		avgDistanceBetweenBricks : REAL;
		brickLength : REAL;
		enableAutoMode : BOOL;
		targetBrickGap : REAL;
		showHighWaitspeedAlarm : BOOL;
		rampUpTime : REAL;
		itemGapTeaching : BOOL;
		enableStaticMode : BOOL;
		showPermanentAutoModeButton : BOOL;
	END_STRUCT;
	hmi_status_FAT_typ : 	STRUCT
		photoSensorTestActive : BOOL; (*Used to open/close dialog in HMI*)
		torqueTestMaxProgress : UDINT;
		torqueTestProgress : UDINT;
		photoSensorTestNoBeltRunning : BOOL;
		photoSensorTestProgress : REAL;
	END_STRUCT;
	local_hw_typ : 	STRUCT
		pwm : {REDUND_UNREPLICABLE} local_hw_pwm_typ; (*Signal name: PWM_BELT
PJ95: M300
Connector: PWM.1
Description: Signal to belt. Motor driver for belt motor*)
		di_photo : BOOL; (*Signal name: DI_CH
PJ95: B300
Connector: DI.01
Description: Signal from Counting head. “1” indicates an element on the belt is passing the counting head*)
	END_STRUCT;
	config_belt_typ : 	STRUCT
		maxTorqueAllowed : REAL := 0.7;
		flickeringFilterGap : REAL := 2.0; (*used when itemGap is disabled*)
		flickeringFilterGapLong : REAL := 4.0; (*used when itemGap is enabled*)
		speedRipple : REAL;
		offsetFromLfCountSpeed : REAL := -20.0;
		hideExperimentalFeatures : BOOL := TRUE;
		brickGapLfMin1Portion : REAL := 35;
		brickGapLfMin2Portion : REAL := 35;
		brickGapLfMin3Portion : REAL := 30;
		brickGapLfMin4Portion : REAL := 30;
		cycleTimeToStopAutoMode1 : REAL := 55;
		cycleTimeToStopAutoMode2 : REAL := 48;
		cycleTimeToStopAutoMode3 : REAL := 43;
		cycleTimeToStopAutoMode4 : REAL := 39;
		brickGapCfMax1Portion : REAL := 130;
		brickGapCfMax2Portion : REAL := 100;
		brickGapCfMax3Portion : REAL := 60;
		brickGapCfMax4Portion : REAL := 52;
		enablePermanentAutoMode : BOOL;
		enableAutoModeFeature : BOOL;
	END_STRUCT;
	recipe_belt_typ : 	STRUCT
		countingSpeed : INT := 300; (*mm/s*)
		waitSpeed : INT := 110; (*mm/s*)
		itemGap : BOOL := FALSE;
		useWaitSpeed : BOOL := TRUE;
		rampUp : INT := 50; (*ms*)
		rampDown : INT := 30; (*ms*)
	END_STRUCT;
	local_alarm_typ : 	STRUCT
		beltBlocked : gAlarm_struct_typ;
		pwmOverVoltage : gAlarm_struct_typ;
		pwmOverTemperature : gAlarm_struct_typ;
		pwmOperatingError : gAlarm_struct_typ;
		pwmCurrentError : gAlarm_struct_typ;
		pwmOverCurrent : gAlarm_struct_typ;
		axisError : gAlarm_struct_typ;
		missingElements : gAlarm_struct_typ;
		pwmModule : gAlarm_struct_typ;
	END_STRUCT;
	local_hw_pwm_typ : 	STRUCT
		periodDuration : UINT;
		pulseWidth : INT;
		clearError : BOOL;
		moduleOk : BOOL;
	END_STRUCT;
END_TYPE
```

#### local.var - Local variables
```iecst
VAR CONSTANT
	MAX_LINEARIZATION_VALUES : USINT := 3;
	INVERSE_COUNT_DIR : USINT := 255;
END_VAR
VAR
	interface : REFERENCE TO gBeltInterface_typ;
	this : {REDUND_UNREPLICABLE} local_typ;
	em : {REDUND_UNREPLICABLE} brdkEM;
	recipe : REFERENCE TO recipe_belt_typ;
	config : REFERENCE TO config_belt_typ;
	axis : {REDUND_UNREPLICABLE} brdkMcBasic;
	j : UINT;
END_VAR
VAR CONSTANT
	MIN_POS_MOVE_AFTER_LAST_BRICK : REAL := 9; (*9mm. (used to avoid that belt stop brick at the end of belt after photosensor)*)
END_VAR
VAR RETAIN
	CFCountSpeed : REAL := 20;
	LFCountSpeed : REAL := 40;
END_VAR
```

#### LocalFunctions.fun
```iecst
FUNCTION_BLOCK BrickGapMeasure
	VAR_INPUT
		Enable : BOOL;
		Signal : {REDUND_UNREPLICABLE} BOOL;
		BeltPosition : REAL;
	END_VAR
	VAR_OUTPUT
		BrickGap : REAL;
	END_VAR
	VAR
		state : USINT;
		lastBeltPosition : REAL;
		totalBrickGap : REAL;
		brickCount : REAL;
	END_VAR
END_FUNCTION_BLOCK

FUNCTION_BLOCK AutoMode
	VAR_INPUT
		Enable : BOOL;
		BeltPosition : REAL;
		BrickGap : REAL;
		BrickCount : UDINT;
		TargetBrickGap : REAL;
	END_VAR
	VAR_OUTPUT
		Measure : BOOL;
		GapOK : BOOL;
		BeltWaitSpeed : REAL;
		CFCountSpeed : REAL;
		CFWaitSpeed : REAL;
		LFCountSpeed : REAL;
		LFWaitSpeed : REAL;
	END_VAR
	VAR
		state : UINT;
		currentBrickCount : UDINT;
		speed : REAL;
		lastBeltPosition : REAL;
		gain : REAL := 0.001;
		totalGapCount : UDINT;
		gapOKCount : UDINT;
	END_VAR
END_FUNCTION_BLOCK

FUNCTION_BLOCK AutoModeSimple
	VAR_INPUT
		Enable : BOOL;
		BrickCount : UDINT := 0;
		BrickGap : REAL;
		TargetBrickGap : REAL;
	END_VAR
	VAR_OUTPUT
		AdjustPercent : SINT;
		GapOK : BOOL;
	END_VAR
	VAR
		currentBrickCount : UDINT;
		state : USINT;
		evaluationCount : UDINT := 15; (*We evalate if we should change adjustPercent every time we count this many bricks*)
		evaluationGap : REAL := 10; (*Target gap +- this variable is accepted*)
	END_VAR
END_FUNCTION_BLOCK

{REDUND_ERROR} FUNCTION_BLOCK BrickInfo (*TODO: Add your comment here*) (*$GROUP=User,$CAT=User,$GROUPICON=User.png,$CATICON=User.png*)
	VAR_INPUT
		Signal : {REDUND_UNREPLICABLE} BOOL;
		Speed : LEGO_SPEED_ENUM;
		BeltPosition : REAL;
		Reset : BOOL;
	END_VAR
	VAR_OUTPUT
		BrickGap : REAL;
		BrickLength : REAL;
		MinBrickGap : REAL;
		BrickGap75 : REAL;
		MissingElements : BOOL;
		BricksTooClosePrc : REAL;
		BrickCount : UDINT;
	END_VAR
	VAR
		state : USINT;
		lastBeltPosition : REAL;
		Median_0 : Median;
		Median_1 : Median;
		Median_MinBrickGap : Median;
		TON_MissingElements : TON;
		MTFilterMovingAverage_0 : MTFilterMovingAverage;
	END_VAR
END_FUNCTION_BLOCK

FUNCTION_BLOCK BrickCounter
	VAR_INPUT
		Signal : BOOL;
		Reset : BOOL;
	END_VAR
	VAR_OUTPUT
		Count : UINT;
		TotalCount : UDINT;
	END_VAR
	VAR
		state : UINT;
		oldReset : BOOL;
	END_VAR
END_FUNCTION_BLOCK

FUNCTION_BLOCK BrickDetector
	VAR_INPUT
		Signal : BOOL;
		ItemGap : {REDUND_UNREPLICABLE} BOOL;
		BeltPosition : REAL;
		FlickeringFilterGap : REAL := 5; (*[mm] Minimum itemgap that is always on til filter flickering of photosensor*)
		FlickeringFilterGapLong : REAL;
	END_VAR
	VAR_OUTPUT
		Teaching : BOOL;
		Out : BOOL;
		BricksCounted : UDINT;
	END_VAR
	VAR
		state : USINT;
		state2 : USINT;
		tmpPosition : REAL;
		lastBeltPosition : REAL;
		avgBrickLength : REAL;
		brickLength : REAL;
		teachingCount : UINT;
		minPosItemGap : REAL := 10;
		tmpPositionFlicker : REAL;
		flickerFilterDist : REAL;
	END_VAR
END_FUNCTION_BLOCK

FUNCTION_BLOCK RampUpTimeCalc
	VAR_INPUT
		Enable : BOOL;
		BeltFeederSensor : BOOL;
		OKPortions : UDINT;
		ChangeOverCounter : UDINT;
		Running : BOOL;
		CFSensor : BOOL := FALSE;
	END_VAR
	VAR_OUTPUT
		RampUpTime : REAL; (*[s]*)
	END_VAR
	VAR
		state : UINT;
		lastChangeOverCounter : UDINT;
		startTime : LREAL;
		lastOKPortions : UDINT;
	END_VAR
END_FUNCTION_BLOCK

FUNCTION_BLOCK Median
	VAR_INPUT
		Reset : BOOL;
		In : REAL;
		BufferLength : UINT := 40;
	END_VAR
	VAR_OUTPUT
		Out : REAL;
		Out75 : REAL;
		Out10 : REAL;
		Out20 : REAL;
	END_VAR
	VAR
		buffer : ARRAY[0..39] OF REAL;
		bufferIdx : UINT;
		tmpBuffer : ARRAY[0..39] OF REAL;
		temp : REAL;
		i : UINT;
		j : UINT;
		noBufferElements : UINT;
	END_VAR
END_FUNCTION_BLOCK

FUNCTION_BLOCK SpeedRippleCalc
	VAR_INPUT
		Enable : BOOL;
		Axis : {REDUND_UNREPLICABLE} UDINT;
	END_VAR
	VAR_OUTPUT
		Out : REAL;
	END_VAR
	VAR
		MC_BR_CyclicRead_0 : MC_BR_CyclicRead;
		MTDataStatistics_0 : MTDataStatistics;
		actVelocity : REAL;
	END_VAR
END_FUNCTION_BLOCK
(*Insert your comment here.*)

FUNCTION_BLOCK PIControllerICM
	VAR_INPUT
		Enable : BOOL;
		Hold : BOOL;
		FreezeIntegral : BOOL;
		IntegralLeak : REAL; (*Makes the integral part leaky*)
		LoopRate : UDINT; (*[ms] loop rate*)
		Setpoint : REAL;
		ProcessValue : REAL;
		Kp : REAL;
		KiNegative : REAL;
		KiPositive : REAL;
		MinOutput : REAL;
		MaxOutput : REAL;
		Integral : REAL;
		Output : REAL;
		FeedForward : REAL;
		InverseControl : BOOL;
	END_VAR
	VAR_OUTPUT
		Active : BOOL;
		Error : REAL;
	END_VAR
	VAR
		state : INT;
		RTInfo_0 : RTInfo;
		loopTime : REAL;
		MaxOutputChange : REAL := 1.0;
		LastOutput : REAL;
	END_VAR
END_FUNCTION_BLOCK

FUNCTION_BLOCK CFController
	VAR_INPUT
		Enable : BOOL;
		StaticOut : REAL;
		Running : BOOL;
		NoElements : BOOL;
		BeltMissingElements : BOOL;
		BrickGap : REAL;
		BrickGapTargetMin : REAL := 40;
		BrickGapTargetMax : REAL;
		MaxOutput : REAL;
		PortionCount : UDINT;
		LFOut : REAL;
		LFOffset : REAL := 10; (*% LF offset to CF output (if 10 then LF will minimum be 10% bigger)*)
	END_VAR
	VAR_OUTPUT
		Active : BOOL;
		Out : REAL;
	END_VAR
	VAR
		state : INT;
		PIControllerICM_0 : PIControllerICM;
		init : BOOL := TRUE;
	END_VAR
END_FUNCTION_BLOCK

FUNCTION_BLOCK LFController
	VAR_INPUT
		Enable : BOOL;
		StaticOut : REAL;
		Running : BOOL;
		NoElements : BOOL;
		BeltMissingElements : BOOL;
		BrickGap : REAL;
		BrickGapTargetMin : REAL := 40;
		BrickGapTargetMax : REAL;
	END_VAR
	VAR_OUTPUT
		Active : BOOL;
		Out : REAL;
	END_VAR
	VAR
		state : INT;
		PIControllerICM_0 : PIControllerICM;
		init : BOOL := TRUE;
	END_VAR
END_FUNCTION_BLOCK

FUNCTION_BLOCK GetBrickGapTargetMinMax
	VAR_INPUT
		PortionCount : UDINT;
	END_VAR
	VAR_OUTPUT
		CFMin : REAL;
		CFMax : REAL;
		LFMin : REAL;
		LFMax : REAL;
	END_VAR
END_FUNCTION_BLOCK

FUNCTION GetBrickGapTargetCF : REAL
	VAR_INPUT
		PortionCount : UDINT;
	END_VAR
END_FUNCTION

FUNCTION GetBrickGapTargetLF : REAL
	VAR_INPUT
		PortionCount : UDINT;
	END_VAR
END_FUNCTION
```

#### LocalFunctions.st
```iecst
(* TODO: Add your comment here *)
FUNCTION_BLOCK BrickDetector
	CASE state OF

		0:
			IF Signal THEN
				Out := TRUE;
				BricksCounted := BricksCounted + 1;
				tmpPosition := BeltPosition;
				flickerFilterDist := SEL(ItemGap,FlickeringFilterGap,FlickeringFilterGapLong); // Use 2 mm extra if itemGap is enabled.
				state := SEL(flickerFilterDist>0.0,30,10);
			END_IF

		10:
			IF NOT Signal THEN
				tmpPositionFlicker := BeltPosition;
				state := 20;
			END_IF

		20:
			IF Signal THEN
				state := 10;
			ELSIF NOT Signal AND ABS(BeltPosition - tmpPositionFlicker) > flickerFilterDist AND ABS(BeltPosition - tmpPosition) > minPosItemGap THEN
				Out := FALSE;
				state := 0;
			END_IF

		30:
			IF NOT Signal THEN
				Out := FALSE;
				state := 0;
			END_IF

	END_CASE

	CASE state2 OF
		0:
			IF ItemGap AND minPosItemGap = 0 THEN
				Teaching := TRUE;
				state2 := 10;
			END_IF
		10:
			IF Signal THEN
				lastBeltPosition := BeltPosition;
				state2 := 20;
			END_IF
		20:
			IF NOT Signal THEN
				brickLength := ABS(BeltPosition-lastBeltPosition);
				teachingCount := teachingCount + 1;
				avgBrickLength := avgBrickLength + brickLength;

				state2 := 10;
				IF teachingCount > 10 THEN
					Teaching := FALSE;
					teachingCount := 0;
					minPosItemGap := avgBrickLength/10.0;
					state2 := 0;
				END_IF
			END_IF
	END_CASE

	IF NOT ItemGap THEN
		minPosItemGap := 0;
		teachingCount := 0;
		avgBrickLength := 0;
		Teaching := FALSE;
		state2 := 0;
	END_IF

END_FUNCTION_BLOCK

FUNCTION_BLOCK BrickInfo
	CASE state OF
		0:
			IF Signal THEN
				state := 10;
			END_IF

		10:
			IF NOT Signal THEN
				Median_0.In := ABS(BeltPosition-lastBeltPosition);
				Median_0();
				lastBeltPosition := BeltPosition;
				state := 20;
			END_IF

		20:
			IF Signal THEN
				Median_1.In := MIN(200, ABS(BeltPosition-lastBeltPosition));
				Median_1();
				Median_MinBrickGap.In := MIN(150, ABS(BeltPosition-lastBeltPosition));
				Median_MinBrickGap();
				lastBeltPosition := BeltPosition;
				TON_MissingElements.IN := FALSE;
				TON_MissingElements();
				BrickCount := BrickCount + 1;
				state := 10;
			END_IF

	END_CASE

	IF BeltPosition < lastBeltPosition THEN
		lastBeltPosition := BeltPosition;
	END_IF

	Median_0.BufferLength := 40;
	Median_1.BufferLength := 20;
	Median_MinBrickGap.BufferLength := 40;

	BrickGap := Median_1.Out;
	MinBrickGap := Median_MinBrickGap.Out20;
	BrickGap75 := Median_MinBrickGap.Out75;
	BrickLength := Median_0.Out75;

	TON_MissingElements.IN := TRUE;
	TON_MissingElements.PT := T#3s;
	TON_MissingElements();

	MissingElements := TON_MissingElements.Q;

	IF Reset THEN
		Reset := FALSE;
		Median_0.Reset := TRUE;
		Median_0();
		Median_1.Reset := TRUE;
		Median_1();
		Median_MinBrickGap.Reset := TRUE;
		Median_MinBrickGap();
		BrickCount := 0;
	END_IF

END_FUNCTION_BLOCK

FUNCTION_BLOCK BrickGapMeasure

	CASE state OF
		0:
			IF Enable THEN
				state := 10;
			END_IF

		10:
			IF Signal THEN
				state := 20;
			END_IF

		20:
			IF NOT Signal THEN
				lastBeltPosition := BeltPosition;
				state := 30;
			END_IF

		30:
			IF Signal THEN
				totalBrickGap := totalBrickGap + LIMIT(0, ABS(BeltPosition-lastBeltPosition), 200);
				brickCount := brickCount + 1;
				BrickGap := totalBrickGap / brickCount;
				state := 20;
			END_IF

	END_CASE

	IF NOT Enable THEN
		totalBrickGap := 0;
		brickCount := 0;
		BrickGap := 0;
		state := 0;
	END_IF

END_FUNCTION_BLOCK

FUNCTION_BLOCK BrickCounter

	CASE state OF
		0:
			IF Signal THEN
				state := 10;
			END_IF

		10:
			IF NOT Signal THEN
				Count := Count + 1;
				TotalCount := TotalCount + 1;
				state := 0;
			END_IF
	END_CASE

	IF Reset AND NOT oldReset THEN
		Count := 0;
	END_IF

	oldReset := Reset;

END_FUNCTION_BLOCK

FUNCTION_BLOCK AutoMode

	CASE state OF
		0:
			IF Enable THEN
				currentBrickCount := BrickCount;
				speed := -0.2;
				BeltWaitSpeed := LIMIT(0, (speed*0.1177+0.288127)*500, 600);
				CFCountSpeed := LIMIT(0, (speed*0.5445+0.334)*87+5, 100);
				CFWaitSpeed := LIMIT(0, (speed*0.357+0.111)*95, 100);
				LFCountSpeed := LIMIT(0, (speed*0.6448+0.31719)*87+13, 100);
				LFWaitSpeed := LIMIT(0, (speed*0.3826+0.1107)*95+5, 100);
				state := 10;
			END_IF

		10: // Wait for new brick
			IF BrickCount > currentBrickCount THEN
				lastBeltPosition := BeltPosition;
				Measure := TRUE;
				state := 20;
			END_IF

		20: // Wait for belt to move
			IF ABS(BeltPosition-lastBeltPosition) > 1000 THEN
				totalGapCount := totalGapCount + 1;
				IF BrickGap = 0 THEN
					speed := speed + 0.01;
					gapOKCount := 0;
				ELSIF ABS(BrickGap - TargetBrickGap) > 5 THEN
					speed := speed + ((BrickGap - TargetBrickGap) * gain);
					gapOKCount := 0;
				ELSE
					gapOKCount := gapOKCount + 1;
				END_IF
				IF gapOKCount > 1 OR totalGapCount > 7 THEN
					GapOK := TRUE;
				END_IF
				BeltWaitSpeed := LIMIT(0, (speed*0.1177+0.288127)*500, 600);
				CFCountSpeed := LIMIT(0, (speed*0.5445+0.334)*87+5, 100);
				CFWaitSpeed := LIMIT(0, (speed*0.357+0.111)*95, 100);
				LFCountSpeed := LIMIT(0, (speed*0.6448+0.31719)*87+13, 100);
				LFWaitSpeed := LIMIT(0, (speed*0.3826+0.1107)*95+5, 100);
				lastBeltPosition := BeltPosition;
				Measure := FALSE;
				state := 30;
			END_IF

		30: // Wait for belt to move to flush bricks
			IF ABS(BeltPosition-lastBeltPosition) > 1000 THEN
				currentBrickCount := BrickCount;
				state := 10;
			END_IF

	END_CASE

	IF NOT Enable AND state <> 0 THEN
		GapOK := FALSE;
		Measure := FALSE;
		state := 0;
	END_IF

END_FUNCTION_BLOCK

FUNCTION_BLOCK AutoModeSimple

	CASE state OF

		0:
			IF Enable THEN
				currentBrickCount := BrickCount;
				AdjustPercent := 0;
				GapOK := FALSE;
				state := 10;
			END_IF

		10:
			IF BrickCount > currentBrickCount + evaluationCount THEN
				currentBrickCount := BrickCount;
				IF BrickGap > TargetBrickGap + evaluationGap AND AdjustPercent < 20 THEN
					AdjustPercent := AdjustPercent + 1;
				ELSIF BrickGap < TargetBrickGap + evaluationGap AND AdjustPercent > -20 THEN
					AdjustPercent := AdjustPercent - 1;
				ELSIF AdjustPercent < 20 AND AdjustPercent > -20 THEN
					// Signal to capcon that we found OK gap
					GapOK := TRUE;
				END_IF
			ELSIF NOT Enable THEN
				AdjustPercent := 0;
				GapOK := FALSE;
				state := 0;
			END_IF

	END_CASE

END_FUNCTION_BLOCK

FUNCTION_BLOCK RampUpTimeCalc

	CASE state OF
		0:
			IF Enable THEN
				lastChangeOverCounter := ChangeOverCounter;
				state := 10;
			END_IF

		10:
			IF ChangeOverCounter <> lastChangeOverCounter AND Running THEN
				lastChangeOverCounter := ChangeOverCounter;
				RampUpTime := 0;
				state := 20;
			END_IF

		20:
			IF BeltFeederSensor OR CFSensor THEN
				startTime := TIME_TO_LREAL(clock_ms());
				lastOKPortions := OKPortions;
				state := 30;
			END_IF

		30:
			IF OKPortions > lastOKPortions THEN
				RampUpTime := LREAL_TO_REAL((TIME_TO_LREAL(clock_ms()) - startTime) / 1000);
				lastChangeOverCounter := ChangeOverCounter;
				state := 10;
			END_IF
	END_CASE

	IF NOT Enable AND state <> 0 THEN
		state := 0;
	END_IF

END_FUNCTION_BLOCK

FUNCTION_BLOCK Median

	buffer[bufferIdx] := In;
	bufferIdx := bufferIdx + 1;
	IF bufferIdx > MIN(SIZEOF(buffer), BufferLength) THEN
		bufferIdx := 0;
	END_IF

	brsmemcpy(ADR(tmpBuffer), ADR(buffer), SIZEOF(tmpBuffer));
	temp := 0;
	FOR i:=0 TO noBufferElements DO
		FOR j:=i+1 TO noBufferElements DO
			IF tmpBuffer[i] > tmpBuffer[j] THEN
				temp := tmpBuffer[i];
				tmpBuffer[i] := tmpBuffer[j];
				tmpBuffer[j] := temp;
			END_IF
		END_FOR
	END_FOR

	noBufferElements := MIN(BufferLength-1, noBufferElements + 1);

	Out10 := tmpBuffer[noBufferElements/10];
	Out20 := tmpBuffer[noBufferElements/5];
	Out := tmpBuffer[noBufferElements/2];
	Out75 := tmpBuffer[noBufferElements*3/5]; // was 3/4

	IF Reset THEN
		Reset := FALSE;
		brsmemset(ADR(buffer), 0, SIZEOF(buffer));
		bufferIdx := 0;
		noBufferElements := 0;
	END_IF

END_FUNCTION_BLOCK

FUNCTION_BLOCK SpeedRippleCalc

	MC_BR_CyclicRead_0.Enable := Enable;
	MC_BR_CyclicRead_0.Axis := Axis;
	MC_BR_CyclicRead_0.DataAddress := ADR(actVelocity);
	MC_BR_CyclicRead_0.DataType := ncPAR_TYP_REAL;
	MC_BR_CyclicRead_0.ParID := ACP10PAR_PCTRL_V_ACT;
	MC_BR_CyclicRead_0();

	MTDataStatistics_0.Enable := Enable AND MC_BR_CyclicRead_0.Valid;
	MTDataStatistics_0.In := ABS(actVelocity/100.0);
	MTDataStatistics_0.MovingWindowLength := 300;
	MTDataStatistics_0();

	Out := 1.28*MTDataStatistics_0.StdDeviation;

END_FUNCTION_BLOCK
```

#### VibratorController.st
```iecst
FUNCTION_BLOCK CFController

	CASE state OF
		0:
			Active := FALSE;
			IF Enable THEN
				Active := TRUE;
				PIControllerICM_0.FeedForward := StaticOut;
				PIControllerICM_0.Output := StaticOut;
				PIControllerICM_0.Integral := 0;
				PIControllerICM_0.Enable := TRUE;
				state := 10;
			ELSE
				Out := StaticOut;
			END_IF

		10:

			// Minimum offset from LF
			IF (PIControllerICM_0.Output+LFOffset) >= LFOut THEN
				Out := LFOut-LFOffset;
				PIControllerICM_0.Hold := TRUE;
			ELSE
				// Check if using a SetPoint interval or not
				IF BrickGapTargetMin <> BrickGapTargetMax THEN
					Out := PIControllerICM_0.Output;
					PIControllerICM_0.Hold := NOT Running OR BeltMissingElements OR NoElements OR (BrickGap >= BrickGapTargetMin AND BrickGap <= BrickGapTargetMax);
				ELSE
					Out := PIControllerICM_0.Output;
					PIControllerICM_0.Hold := NOT Running OR BeltMissingElements OR NoElements;
				END_IF
			END_IF

			IF NOT Enable THEN
				PIControllerICM_0.Enable := FALSE;
				state := 0;
			END_IF

	END_CASE

	IF init THEN
		init := FALSE;
		PIControllerICM_0.InverseControl := TRUE;
		PIControllerICM_0.Kp := 0.011;
		PIControllerICM_0.KiPositive := 0.011;
		PIControllerICM_0.KiNegative := 0.011;
		PIControllerICM_0.LoopRate := 1000;
		PIControllerICM_0.MinOutput := 5;
		PIControllerICM_0.IntegralLeak := 0.05;
		PIControllerICM_0.Hold := TRUE;
	END_IF

	PIControllerICM_0.ProcessValue := BrickGap;
	PIControllerICM_0.Setpoint := BrickGapTargetMin;
	PIControllerICM_0.MaxOutput := MaxOutput;
	PIControllerICM_0();

END_FUNCTION_BLOCK

FUNCTION_BLOCK LFController

	CASE state OF
		0:
			Active := FALSE;
			IF Enable THEN
				Active := TRUE;
				PIControllerICM_0.FeedForward := StaticOut;
				PIControllerICM_0.Output := StaticOut;
				PIControllerICM_0.Integral := 0;
				PIControllerICM_0.Enable := TRUE;
				state := 10;
			ELSE
				Out := StaticOut;
			END_IF

		10:
			// Check if using a SetPoint interval or not
			IF BrickGapTargetMin <> BrickGapTargetMax THEN
				PIControllerICM_0.Hold := NOT Running OR BeltMissingElements OR (BrickGap >= BrickGapTargetMin AND BrickGap <= BrickGapTargetMax);
			ELSE
				PIControllerICM_0.Hold := NOT Running OR BeltMissingElements;
			END_IF

			Out := PIControllerICM_0.Output;

			IF NOT Enable THEN
				PIControllerICM_0.Enable := FALSE;
				state := 0;
			END_IF

	END_CASE

	IF init THEN
		init := FALSE;
		PIControllerICM_0.InverseControl := TRUE;
		PIControllerICM_0.Kp := 0.015;
		PIControllerICM_0.KiPositive := 0.015;
		PIControllerICM_0.KiNegative := 0.015;
		PIControllerICM_0.LoopRate := 1000;
		PIControllerICM_0.MinOutput := 10;
		PIControllerICM_0.MaxOutput := 130;
		PIControllerICM_0.IntegralLeak := 0.05;
		PIControllerICM_0.Hold := TRUE;
	END_IF

	PIControllerICM_0.ProcessValue := BrickGap;
	PIControllerICM_0.Setpoint := BrickGapTargetMin;
	PIControllerICM_0();

END_FUNCTION_BLOCK

FUNCTION_BLOCK PIControllerICM

	IF NOT Enable AND Active THEN
		state := 0;
		Error := 0;
		Integral := 0;
		Output := 0;
		loopTime := 0;
		Active := FALSE;
	END_IF

	CASE state OF
		0:
			IF Enable THEN
				Active := TRUE;
				state := 10;
			END_IF

		10:
			RTInfo_0.enable := TRUE;
			RTInfo_0();

			IF RTInfo_0.status = ERR_OK THEN
				LastOutput := Output;
				state := 20;
			END_IF

		20:

			loopTime := loopTime + RTInfo_0.cycle_time / 1000;

			IF loopTime >= LoopRate THEN
				loopTime := 0;

				IF NOT Hold THEN

					// Calculate the error
					IF InverseControl THEN
						Error := ProcessValue - Setpoint;
					ELSE
						Error := Setpoint - ProcessValue;
					END_IF

					// Anti windup if output is saturated
					IF ((Output > MinOutput AND Output < MaxOutput) OR (Output = MinOutput AND Error > 0) OR (Output = MaxOutput AND Error < 0)) AND NOT FreezeIntegral THEN
						// Integral accumulation
						IF Error > 0 THEN
							Integral := Integral + (KiPositive * Error);
						ELSE
							Integral := Integral + (KiNegative * Error);
						END_IF

						Integral := Integral - IntegralLeak;
					END_IF

					// PI controller formula with limits on output
					Output := LIMIT(MinOutput, Kp * Error + Integral + FeedForward, MaxOutput);

					// Rate limiting to prevent sudden large changes
					IF Output > LastOutput + MaxOutputChange THEN
						Output := LastOutput + MaxOutputChange;
					ELSIF Output < LastOutput - MaxOutputChange THEN
						Output := LastOutput - MaxOutputChange;
					END_IF
					LastOutput := Output;

				ELSE
				//	Integral := Integral - IntegralLeak;
				END_IF
			END_IF
	END_CASE

END_FUNCTION_BLOCK

FUNCTION_BLOCK GetBrickGapTargetMinMax
	(* Get SetPoint interval *)
	CASE PortionCount OF

		0,1:
			CFMin := 55;
			CFMax := 130;
			LFMin := 35;
			LFMax := 70;

		2:
			CFMin := 55;
			CFMax := 100;
			LFMin := 35;
			LFMax := 45;

		3:
			CFMin := 50;
			CFMax := 60;
			LFMin := 30;
			LFMax := 30;

		4:
			CFMin := 50;
			CFMax := 55;
			LFMin := 30;
			LFMax := 30;

		ELSE
			CFMin := 55;
			CFMax := 55;
			LFMin := 30;
			LFMax := 30;

	END_CASE

END_FUNCTION_BLOCK

FUNCTION GetBrickGapTargetCF
	CASE PortionCount OF
		0,1:
			GetBrickGapTargetCF := 100;
		2:
			GetBrickGapTargetCF := 80;
		3:
			GetBrickGapTargetCF := 60;
		4:
			GetBrickGapTargetCF := 55;
		ELSE
			GetBrickGapTargetCF := 55;
	END_CASE
END_FUNCTION

FUNCTION GetBrickGapTargetLF
	CASE PortionCount OF
		0,1:
			GetBrickGapTargetLF := 60;
		2:
			GetBrickGapTargetLF := 50;
		3:
			GetBrickGapTargetLF := 40;
		4:
			GetBrickGapTargetLF := 35;
		ELSE
			GetBrickGapTargetLF := 35;
	END_CASE
END_FUNCTION
```

### beltGlobal.typ
```iecst
TYPE
	gBeltInterface_typ : 	STRUCT
		cmd : gBeltInterface_cmd_typ;
		status : gBeltInterface_status_typ;
		parameter : gBeltInterface_par_typ;
	END_STRUCT;
	gBeltInterface_cmd_typ : 	STRUCT
		count : BOOL;
		calibrate : BOOL;
		dropBrick : BOOL;
		emptyStop : BOOL;
		capconTimeOut : BOOL; (*capcon -> belt. Belt signaled that capcon should get a brick but it never arrived, signal back to belt that the brick never arrived.*)
		copyRecipe : copy_recipe_command_typ;
		afterCount : BOOL; (*capcon -> belt. We just had an aftercount*)
		runManualTest : BOOL;
		putRecipeForStalkElement : BOOL;
		initRecipe : BOOL;
		changeover : BOOL; (*vibrator -> belt. We have changeover and recipe values has been updated.*)
		cycleTimeCount : UDINT;
		stopDoingEmpty : BOOL;
		setDirection : BOOL;
		doPhotoSensorTest : BOOL;
		doPhotoSensorTestNoBelt : BOOL;
		doTorqueTest : BOOL;
	END_STRUCT;
	gBeltInterface_par_typ : 	STRUCT
		brickCountInPortion : UDINT;
		speedManualTest : REAL;
		direction : USINT;
	END_STRUCT;
	gBeltInterface_status_typ : 	STRUCT
		running : BOOL; (*The belt is moving*)
		countingDone : BOOL;
		teachingDone : BOOL;
		speed : LEGO_SPEED_ENUM;
		calibratingMode : BOOL;
		bricksInPortion : INT;
		useVibratorWaitSpeed : BOOL;
		dropBrickDone : BOOL;
		adjustPercent : SINT;
		autoMode : BOOL;
		CFCountSpeed : REAL;
		CFWaitSpeed : REAL;
		LFCountSpeed : REAL;
		LFWaitSpeed : REAL;
		gapOK : BOOL;
		autoModeSimple : BOOL;
		actualPosition : REAL;
		recipeLoaded : BOOL;
		photoSensorTestResult : testResult_enum;
		torqueTestTestResult : testResult_enum;
		photoSensorTestNoBeltResult : testResult_enum;
	END_STRUCT;
	testResult_enum :
		( (*Enum to get feedback if test is OK or NOK*)
		TEST_NOT_DONE := 0,
		TEST_OK := 1,
		TEST_NOT_OK := 2,
		TEST_STOPPED := 3
		);
END_TYPE
```

### beltGlobal.var
```iecst
VAR
	gBeltInterface : gBeltInterface_typ;
END_VAR
```

### Program Logical/modules/main/capcon/capcon (IEC)
